C07325=1163.883,398.048,-85.044,-176.099,9.432,148.794
C07326=1163.887,397.800,-85.007,-176.099,9.430,148.793
C07327=1163.891,397.553,-84.971,-176.098,9.427,148.792
C07328=1163.895,397.306,-84.934,-176.097,9.426,148.792
C07329=1163.898,397.058,-84.899,-176.097,9.423,148.791
C07330=1163.903,396.811,-84.862,-176.097,9.420,148.790
C07331=1163.906,396.564,-84.826,-176.097,9.418,148.789
C07332=1163.910,396.316,-84.790,-176.096,9.416,148.789
C07333=1163.914,396.069,-84.754,-176.095,9.413,148.788
C07334=1163.918,395.822,-84.717,-176.095,9.410,148.787
C07335=1163.922,395.575,-84.680,-176.095,9.408,148.786
C07336=1163.926,395.327,-84.645,-176.094,9.406,148.785
C07337=1163.930,395.080,-84.608,-176.094,9.403,148.785
C07338=1163.934,394.832,-84.572,-176.094,9.401,148.784
C07339=1163.938,394.585,-84.535,-176.093,9.398,148.783
C07340=1163.941,394.338,-84.500,-176.093,9.395,148.782
C07341=1163.945,394.090,-84.463,-176.093,9.393,148.782
C07342=1163.949,393.843,-84.428,-176.092,9.390,148.781
C07343=1163.953,393.596,-84.391,-176.092,9.387,148.780
C07344=1163.957,393.349,-84.354,-176.091,9.385,148.779
C07345=1163.961,393.101,-84.318,-176.091,9.383,148.779
C07346=1163.964,392.854,-84.282,-176.091,9.379,148.778
C07347=1163.969,392.606,-84.246,-176.091,9.377,148.777
C07348=1163.972,392.359,-84.210,-176.091,9.374,148.776
C07349=1163.976,392.112,-84.173,-176.090,9.371,148.775
C07350=1163.980,391.827,-84.131,-176.090,9.368,148.775
C07351=1163.985,391.541,-84.090,-176.090,9.365,148.774
C07352=1163.990,391.256,-84.048,-176.089,9.362,148.773
C07353=1163.994,390.970,-84.006,-176.090,9.358,148.772
C07354=1163.998,390.723,-83.971,-176.089,9.355,148.771
C07355=1164.002,390.476,-83.934,-176.089,9.353,148.770
C07356=1164.006,390.228,-83.898,-176.089,9.349,148.770
C07357=1164.010,389.981,-83.861,-176.089,9.347,148.769
C07358=1164.013,389.733,-83.826,-176.089,9.344,148.768
C07359=1164.018,389.486,-83.789,-176.089,9.341,148.767
C07360=1164.021,389.239,-83.753,-176.089,9.338,148.766
C07361=1164.025,388.992,-83.717,-176.088,9.335,148.766
C07362=1164.029,388.744,-83.681,-176.089,9.332,148.765
C07363=1164.033,388.497,-83.644,-176.089,9.329,148.764
C07364=1164.037,388.249,-83.609,-176.089,9.326,148.763
C07365=1164.041,388.002,-83.572,-176.090,9.322,148.763
C07366=1164.044,387.755,-83.536,-176.089,9.320,148.762
C07367=1164.048,387.507,-83.501,-176.089,9.316,148.761
C07368=1164.052,387.260,-83.464,-176.090,9.313,148.760
C07369=1164.056,387.013,-83.428,-176.090,9.310,148.759
C07370=1164.060,386.765,-83.391,-176.090,9.307,148.759
C07371=1164.064,386.518,-83.356,-176.091,9.303,148.758
C07372=1164.068,386.270,-83.320,-176.091,9.300,148.757
C07373=1164.072,386.024,-83.284,-176.091,9.297,148.756
C07374=1164.076,385.776,-83.248,-176.091,9.294,148.756
C07375=1164.080,385.529,-83.211,-176.092,9.291,148.755
C07376=1164.083,385.282,-83.176,-176.092,9.287,148.754
C07377=1164.088,385.034,-83.140,-176.093,9.284,148.753
C07378=1164.091,384.787,-83.103,-176.093,9.281,148.753
C07379=1164.096,384.539,-83.067,-176.094,9.277,148.752
C07380=1164.099,384.292,-83.032,-176.094,9.274,148.751
C07381=1164.103,384.045,-82.996,-176.095,9.271,148.750
C07382=1164.107,383.797,-82.959,-176.096,9.266,148.750
C07383=1164.111,383.549,-82.924,-176.096,9.263,148.749
C07384=1164.114,383.303,-82.888,-176.097,9.260,148.748
C07385=1164.118,383.055,-82.851,-176.098,9.257,148.747
C07386=1164.123,382.808,-82.816,-176.099,9.252,148.747
C07387=1164.127,382.560,-82.780,-176.099,9.249,148.746
C07388=1164.130,382.313,-82.744,-176.100,9.246,148.745
C07389=1164.134,382.066,-82.708,-176.100,9.243,148.745
C07390=1164.139,381.818,-82.672,-176.101,9.238,148.744
C07391=1164.142,381.570,-82.637,-176.102,9.235,148.743
C07392=1164.146,381.324,-82.600,-176.103,9.231,148.742
C07393=1164.150,381.076,-82.564,-176.104,9.228,148.742
C07394=1164.154,380.828,-82.529,-176.105,9.224,148.741
C07395=1164.157,380.581,-82.493,-176.106,9.221,148.740
C07396=1164.162,380.334,-82.457,-176.107,9.217,148.740
C07397=1164.166,380.087,-82.421,-176.108,9.213,148.739
C07398=1164.169,379.839,-82.385,-176.109,9.209,148.738
C07399=1164.173,379.592,-82.350,-176.110,9.206,148.738
C07400=1164.177,379.344,-82.314,-176.111,9.202,148.737
C07401=1164.181,379.096,-82.278,-176.113,9.198,148.736
C07402=1164.185,378.849,-82.243,-176.113,9.195,148.736
C07403=1164.190,378.602,-82.207,-176.115,9.191,148.735
C07404=1164.193,378.355,-82.171,-176.116,9.187,148.734
C07405=1164.197,378.107,-82.135,-176.117,9.184,148.734
C07406=1164.200,377.860,-82.100,-176.118,9.180,148.733
C07407=1164.205,377.612,-82.063,-176.120,9.176,148.732
C07408=1164.208,377.365,-82.028,-176.121,9.172,148.732
C07409=1164.213,377.118,-81.993,-176.122,9.168,148.731
C07410=1164.216,376.870,-81.957,-176.123,9.165,148.731
C07411=1164.220,376.623,-81.922,-176.125,9.161,148.730
C07412=1164.224,376.375,-81.885,-176.126,9.157,148.729
C07413=1164.228,376.128,-81.850,-176.128,9.154,148.729
C07414=1164.232,375.881,-81.815,-176.129,9.150,148.728
C07415=1164.236,375.633,-81.779,-176.131,9.146,148.728
C07416=1164.240,375.386,-81.744,-176.132,9.142,148.727
C07417=1164.244,375.138,-81.707,-176.134,9.138,148.726
C07418=1164.248,374.890,-81.672,-176.136,9.135,148.726
C07419=1164.252,374.644,-81.637,-176.137,9.131,148.725
C07420=1164.256,374.396,-81.601,-176.138,9.127,148.725
C07421=1164.259,374.149,-81.566,-176.140,9.123,148.724
C07422=1164.263,373.901,-81.530,-176.142,9.119,148.724
C07423=1164.267,373.653,-81.495,-176.144,9.116,148.723
C07424=1164.272,373.406,-81.460,-176.145,9.112,148.723
C07425=1164.276,373.158,-81.424,-176.147,9.108,148.722
C07426=1164.279,372.911,-81.388,-176.148,9.104,148.722
C07427=1164.283,372.663,-81.353,-176.150,9.101,148.721
C07428=1164.287,372.417,-81.318,-176.152,9.097,148.721
C07429=1164.291,372.169,-81.282,-176.154,9.092,148.720
C07430=1164.295,371.921,-81.247,-176.156,9.089,148.720
C07431=1164.299,371.674,-81.212,-176.157,9.085,148.719
C07432=1164.303,371.427,-81.177,-176.159,9.081,148.719
C07433=1164.306,371.179,-81.141,-176.161,9.078,148.718
C07434=1164.310,370.931,-81.106,-176.163,9.073,148.717
C07435=1164.315,370.684,-81.071,-176.165,9.069,148.717
C07436=1164.318,370.437,-81.035,-176.167,9.066,148.717
C07437=1164.322,370.189,-81.000,-176.169,9.062,148.716
C07438=1164.327,369.942,-80.965,-176.171,9.059,148.716
C07439=1164.330,369.694,-80.930,-176.173,9.054,148.715
C07440=1164.334,369.447,-80.894,-176.175,9.051,148.715
C07441=1164.338,369.199,-80.860,-176.176,9.047,148.714
C07442=1164.342,368.952,-80.824,-176.179,9.042,148.714
C07443=1164.346,368.704,-80.789,-176.181,9.039,148.713
C07444=1164.350,368.456,-80.754,-176.182,9.035,148.713
C07445=1164.354,368.210,-80.719,-176.185,9.031,148.713
C07446=1164.358,367.961,-80.684,-176.187,9.027,148.712
C07447=1164.362,367.714,-80.648,-176.189,9.024,148.712
C07448=1164.366,367.467,-80.613,-176.191,9.019,148.711
C07449=1164.370,367.219,-80.578,-176.193,9.016,148.711
C07450=1164.374,366.972,-80.543,-176.195,9.012,148.710
C07451=1164.378,366.724,-80.508,-176.198,9.008,148.710
C07452=1164.382,366.477,-80.473,-176.200,9.004,148.710
C07453=1164.386,366.229,-80.438,-176.202,9.001,148.709
C07454=1164.391,365.947,-80.399,-176.204,8.996,148.709
C07455=1164.395,365.664,-80.359,-176.207,8.992,148.708
C07456=1164.399,365.382,-80.319,-176.209,8.988,148.708
C07457=1164.403,365.100,-80.279,-176.212,8.983,148.707
C07458=1164.407,364.852,-80.244,-176.214,8.979,148.707
C07459=1164.412,364.605,-80.209,-176.216,8.975,148.707
C07460=1164.416,364.357,-80.174,-176.219,8.971,148.706
C07461=1164.420,364.110,-80.139,-176.221,8.968,148.706
C07462=1164.423,363.862,-80.105,-176.223,8.964,148.706
C07463=1164.427,363.614,-80.070,-176.226,8.960,148.705
C07464=1164.431,363.367,-80.035,-176.228,8.956,148.705
C07465=1164.435,363.119,-80.000,-176.231,8.952,148.705
C07466=1164.440,362.872,-79.965,-176.232,8.949,148.704
C07467=1164.443,362.624,-79.931,-176.235,8.945,148.704
C07468=1164.447,362.377,-79.896,-176.237,8.941,148.704
C07469=1164.451,362.129,-79.861,-176.239,8.938,148.703
C07470=1164.455,361.881,-79.826,-176.242,8.933,148.703
C07471=1164.459,361.634,-79.792,-176.244,8.930,148.703
C07472=1164.463,361.386,-79.757,-176.247,8.926,148.702
C07473=1164.467,361.139,-79.723,-176.249,8.922,148.702
C07474=1164.471,360.891,-79.688,-176.251,8.918,148.701
C07475=1164.475,360.643,-79.654,-176.254,8.915,148.701
C07476=1164.479,360.396,-79.618,-176.256,8.910,148.701
C07477=1164.483,360.149,-79.584,-176.258,8.907,148.701
C07478=1164.487,359.901,-79.550,-176.261,8.904,148.700
C07479=1164.491,359.653,-79.515,-176.263,8.899,148.700
C07480=1164.494,359.406,-79.481,-176.265,8.896,148.700
C07481=1164.499,359.158,-79.446,-176.268,8.892,148.699
C07482=1164.503,358.910,-79.412,-176.270,8.888,148.699
C07483=1164.507,358.663,-79.378,-176.273,8.884,148.699
C07484=1164.511,358.415,-79.343,-176.275,8.881,148.698
C07485=1164.515,358.168,-79.309,-176.277,8.877,148.698
C07486=1164.519,357.921,-79.274,-176.280,8.873,148.698
C07487=1164.523,357.673,-79.239,-176.282,8.870,148.698
C07488=1164.527,357.426,-79.205,-176.285,8.866,148.697
C07489=1164.531,357.178,-79.170,-176.287,8.862,148.697
C07490=1164.535,356.930,-79.137,-176.289,8.859,148.697
C07491=1164.539,356.682,-79.102,-176.292,8.855,148.696
C07492=1164.543,356.435,-79.068,-176.294,8.851,148.696
C07493=1164.547,356.187,-79.034,-176.297,8.847,148.696
C07494=1164.550,355.939,-79.000,-176.299,8.844,148.695
C07495=1164.555,355.692,-78.965,-176.302,8.840,148.695
C07496=1164.558,355.444,-78.931,-176.304,8.836,148.695
C07497=1164.563,355.197,-78.897,-176.306,8.833,148.695
C07498=1164.567,354.950,-78.863,-176.309,8.829,148.694
C07499=1164.571,354.701,-78.828,-176.311,8.825,148.694
C07500=1164.575,354.454,-78.795,-176.313,8.822,148.694
C07501=1164.579,354.206,-78.760,-176.316,8.817,148.693
C07502=1164.583,353.958,-78.726,-176.318,8.814,148.693
C07503=1164.587,353.711,-78.692,-176.321,8.811,148.693
C07504=1164.590,353.463,-78.657,-176.323,8.806,148.693
C07505=1164.595,353.215,-78.624,-176.325,8.803,148.692
C07506=1164.599,352.968,-78.590,-176.328,8.800,148.692
C07507=1164.602,352.720,-78.555,-176.331,8.796,148.692
C07508=1164.607,352.473,-78.521,-176.333,8.792,148.692
C07509=1164.611,352.225,-78.488,-176.335,8.789,148.691
C07510=1164.615,351.977,-78.453,-176.338,8.785,148.691
C07511=1164.619,351.730,-78.419,-176.340,8.781,148.691
C07512=1164.623,351.482,-78.386,-176.342,8.778,148.690
C07513=1164.627,351.235,-78.351,-176.345,8.774,148.690
C07514=1164.631,350.987,-78.317,-176.347,8.771,148.690
C07515=1164.635,350.739,-78.284,-176.350,8.766,148.690
C07516=1164.639,350.492,-78.250,-176.352,8.763,148.689
C07517=1164.643,350.243,-78.216,-176.354,8.760,148.689
C07518=1164.647,349.996,-78.182,-176.357,8.756,148.689
C07519=1164.652,349.748,-78.148,-176.360,8.752,148.689
C07520=1164.656,349.501,-78.115,-176.362,8.749,148.688
C07521=1164.659,349.253,-78.080,-176.365,8.745,148.688
C07522=1164.664,349.005,-78.047,-176.367,8.742,148.688
C07523=1164.667,348.758,-78.013,-176.369,8.738,148.688
C07524=1164.672,348.510,-77.980,-176.372,8.734,148.687
C07525=1164.676,348.262,-77.945,-176.374,8.731,148.687
C07526=1164.680,348.015,-77.912,-176.376,8.727,148.687
C07527=1164.684,347.767,-77.878,-176.379,8.724,148.687
C07528=1164.688,347.520,-77.845,-176.382,8.720,148.686
C07529=1164.691,347.271,-77.811,-176.384,8.717,148.686
C07530=1164.696,347.024,-77.777,-176.386,8.713,148.686
C07531=1164.700,346.776,-77.743,-176.389,8.709,148.686
C07532=1164.704,346.528,-77.710,-176.391,8.706,148.685
C07533=1164.708,346.281,-77.676,-176.394,8.703,148.685
C07534=1164.712,346.033,-77.642,-176.396,8.699,148.685
C07535=1164.716,345.785,-77.608,-176.399,8.695,148.685
C07536=1164.720,345.538,-77.575,-176.401,8.692,148.685
C07537=1164.724,345.290,-77.542,-176.403,8.688,148.684
C07538=1164.728,345.042,-77.509,-176.406,8.684,148.684
C07539=1164.732,344.795,-77.475,-176.408,8.681,148.684
C07540=1164.736,344.547,-77.442,-176.410,8.678,148.684
C07541=1164.741,344.299,-77.408,-176.413,8.674,148.683
C07542=1164.745,344.051,-77.375,-176.416,8.670,148.683
C07543=1164.749,343.804,-77.341,-176.418,8.667,148.683
C07544=1164.753,343.556,-77.308,-176.421,8.663,148.683
C07545=1164.757,343.308,-77.274,-176.423,8.660,148.682
C07546=1164.761,343.061,-77.241,-176.425,8.656,148.682
C07547=1164.765,342.813,-77.208,-176.428,8.652,148.682
C07548=1164.768,342.565,-77.174,-176.430,8.649,148.682
C07549=1164.773,342.317,-77.141,-176.433,8.646,148.681
C07550=1164.777,342.070,-77.108,-176.435,8.642,148.681
C07551=1164.781,341.822,-77.074,-176.438,8.638,148.681
C07552=1164.786,341.574,-77.041,-176.441,8.635,148.681
C07553=1164.790,341.326,-77.008,-176.443,8.632,148.681
C07554=1164.794,341.078,-76.974,-176.445,8.629,148.681
C07555=1164.798,340.831,-76.941,-176.448,8.624,148.680
C07556=1164.802,340.583,-76.908,-176.450,8.621,148.680
C07557=1164.806,340.335,-76.875,-176.453,8.618,148.680
C07558=1164.811,340.056,-76.837,-176.456,8.614,148.680
C07559=1164.815,339.776,-76.800,-176.458,8.610,148.679
C07560=1164.819,339.497,-76.763,-176.461,8.606,148.679
C07561=1164.824,339.217,-76.725,-176.464,8.602,148.679
C07562=1164.828,338.970,-76.692,-176.466,8.598,148.679
C07563=1164.832,338.722,-76.659,-176.469,8.595,148.678
C07564=1164.836,338.474,-76.626,-176.471,8.592,148.678
C07565=1164.841,338.226,-76.593,-176.474,8.587,148.678
C07566=1164.845,337.979,-76.560,-176.476,8.584,148.678
C07567=1164.849,337.730,-76.527,-176.479,8.581,148.678
C07568=1164.853,337.483,-76.494,-176.481,8.578,148.678
C07569=1164.857,337.235,-76.461,-176.484,8.574,148.677
C07570=1164.861,336.987,-76.428,-176.486,8.570,148.677
C07571=1164.865,336.740,-76.395,-176.489,8.567,148.677
C07572=1164.869,336.492,-76.362,-176.491,8.564,148.677
C07573=1164.874,336.244,-76.330,-176.493,8.561,148.677
C07574=1164.878,335.996,-76.296,-176.496,8.556,148.676
C07575=1164.882,335.748,-76.263,-176.499,8.553,148.676
C07576=1164.885,335.501,-76.231,-176.501,8.550,148.676
C07577=1164.890,335.252,-76.198,-176.503,8.547,148.676
C07578=1164.894,335.005,-76.165,-176.506,8.543,148.676
C07579=1164.898,334.757,-76.132,-176.509,8.540,148.675
C07580=1164.901,334.509,-76.099,-176.511,8.536,148.675
C07581=1164.906,334.261,-76.067,-176.513,8.533,148.675
C07582=1164.910,334.013,-76.034,-176.517,8.529,148.675
C07583=1164.914,333.766,-76.001,-176.519,8.526,148.675
C07584=1164.918,333.518,-75.969,-176.521,8.523,148.675
C07585=1164.922,333.270,-75.936,-176.523,8.519,148.674
C07586=1164.926,333.022,-75.902,-176.526,8.516,148.674
C07587=1164.931,332.774,-75.870,-176.529,8.512,148.674
C07588=1164.935,332.527,-75.838,-176.531,8.509,148.674
C07589=1164.939,332.279,-75.805,-176.534,8.506,148.674
C07590=1164.943,332.031,-75.772,-176.536,8.502,148.674
C07591=1164.947,331.783,-75.740,-176.539,8.498,148.673
C07592=1164.951,331.535,-75.707,-176.541,8.495,148.673
C07593=1164.955,331.287,-75.675,-176.544,8.492,148.673
C07594=1164.959,331.039,-75.642,-176.546,8.489,148.673
C07595=1164.963,330.791,-75.610,-176.548,8.485,148.673
C07596=1164.967,330.543,-75.577,-176.551,8.481,148.672
C07597=1164.972,330.296,-75.545,-176.554,8.478,148.672
C07598=1164.976,330.048,-75.512,-176.556,8.475,148.672
C07599=1164.980,329.800,-75.480,-176.559,8.472,148.672
C07600=1164.984,329.553,-75.447,-176.561,8.468,148.672
C07601=1164.988,329.304,-75.415,-176.564,8.464,148.672
C07602=1164.991,329.057,-75.382,-176.566,8.461,148.672
C07603=1164.997,328.809,-75.350,-176.569,8.458,148.671
C07604=1165.001,328.561,-75.317,-176.571,8.455,148.671
C07605=1165.004,328.313,-75.285,-176.573,8.451,148.671
C07606=1165.009,328.065,-75.252,-176.577,8.448,148.671
C07607=1165.013,327.817,-75.221,-176.579,8.444,148.671
C07608=1165.017,327.570,-75.188,-176.581,8.441,148.671
C07609=1165.021,327.322,-75.156,-176.584,8.438,148.670
C07610=1165.025,327.074,-75.124,-176.586,8.435,148.670
C07611=1165.029,326.826,-75.091,-176.589,8.431,148.670
C07612=1165.033,326.578,-75.059,-176.591,8.427,148.670
C07613=1165.038,326.330,-75.027,-176.594,8.424,148.670
C07614=1165.042,326.082,-74.995,-176.597,8.421,148.670
C07615=1165.046,325.834,-74.963,-176.599,8.418,148.670
C07616=1165.050,325.586,-74.930,-176.601,8.414,148.669
C07617=1165.054,325.339,-74.898,-176.604,8.412,148.669
C07618=1165.059,325.091,-74.866,-176.607,8.407,148.669
C07619=1165.062,324.843,-74.834,-176.609,8.404,148.669
C07620=1165.066,324.595,-74.802,-176.612,8.401,148.669
C07621=1165.071,324.347,-74.770,-176.614,8.398,148.669
C07622=1165.074,324.100,-74.737,-176.616,8.395,148.668
C07623=1165.079,323.851,-74.705,-176.619,8.392,148.668
C07624=1165.083,323.603,-74.673,-176.622,8.387,148.668
C07625=1165.087,323.356,-74.642,-176.624,8.384,148.668
C07626=1165.091,323.107,-74.609,-176.627,8.381,148.668
C07627=1165.095,322.859,-74.577,-176.629,8.378,148.668
C07628=1165.099,322.612,-74.546,-176.632,8.375,148.668
C07629=1165.104,322.364,-74.513,-176.634,8.372,148.668
C07630=1165.108,322.116,-74.482,-176.637,8.368,148.667
C07631=1165.111,321.868,-74.450,-176.639,8.364,148.667
C07632=1165.116,321.620,-74.418,-176.642,8.361,148.667
C07633=1165.120,321.372,-74.386,-176.644,8.358,148.667
C07634=1165.124,321.124,-74.354,-176.647,8.355,148.667
C07635=1165.129,320.876,-74.322,-176.650,8.352,148.667
C07636=1165.132,320.628,-74.290,-176.652,8.348,148.667
C07637=1165.136,320.380,-74.258,-176.655,8.344,148.666
C07638=1165.140,320.133,-74.227,-176.657,8.341,148.666
C07639=1165.145,319.885,-74.194,-176.660,8.338,148.666
C07640=1165.149,319.636,-74.162,-176.662,8.335,148.666
C07641=1165.153,319.389,-74.132,-176.665,8.332,148.666
C07642=1165.157,319.140,-74.100,-176.667,8.328,148.666
C07643=1165.162,318.893,-74.068,-176.670,8.326,148.666
C07644=1165.166,318.645,-74.036,-176.673,8.321,148.666
C07645=1165.169,318.397,-74.004,-176.675,8.318,148.665
C07646=1165.174,318.149,-73.973,-176.678,8.315,148.665
C07647=1165.178,317.901,-73.941,-176.680,8.312,148.665
C07648=1165.183,317.653,-73.909,-176.683,8.309,148.665
C07649=1165.186,317.405,-73.878,-176.685,8.306,148.665
C07650=1165.190,317.157,-73.846,-176.687,8.302,148.665
C07651=1165.195,316.909,-73.815,-176.690,8.299,148.665
C07652=1165.198,316.661,-73.783,-176.693,8.295,148.665
C07653=1165.203,316.414,-73.752,-176.696,8.292,148.665
C07654=1165.208,316.165,-73.720,-176.698,8.289,148.665
C07655=1165.212,315.917,-73.688,-176.700,8.286,148.664
C07656=1165.216,315.669,-73.657,-176.703,8.283,148.664
C07657=1165.220,315.421,-73.625,-176.705,8.279,148.664
C07658=1165.224,315.173,-73.594,-176.708,8.276,148.664
C07659=1165.228,314.925,-73.562,-176.710,8.273,148.664
C07660=1165.232,314.677,-73.531,-176.714,8.269,148.664
C07661=1165.236,314.429,-73.499,-176.716,8.266,148.664
C07662=1165.241,314.152,-73.464,-176.719,8.263,148.664
C07663=1165.246,313.875,-73.430,-176.722,8.259,148.664
C07664=1165.250,313.598,-73.394,-176.724,8.256,148.664
C07665=1165.255,313.321,-73.359,-176.727,8.252,148.663
C07666=1165.259,313.073,-73.329,-176.729,8.249,148.663
C07667=1165.263,312.825,-73.297,-176.732,8.246,148.663
C07668=1165.267,312.577,-73.266,-176.734,8.242,148.663
C07669=1165.271,312.329,-73.234,-176.737,8.239,148.663
C07670=1165.276,312.081,-73.203,-176.740,8.235,148.663
C07671=1165.280,311.833,-73.172,-176.743,8.232,148.663
C07672=1165.284,311.585,-73.141,-176.745,8.229,148.663
C07673=1165.288,311.337,-73.109,-176.748,8.226,148.663
C07674=1165.292,311.089,-73.078,-176.750,8.223,148.662
C07675=1165.296,310.840,-73.047,-176.753,8.220,148.662
C07676=1165.301,310.593,-73.016,-176.755,8.216,148.662
C07677=1165.305,310.345,-72.985,-176.758,8.213,148.662
C07678=1165.309,310.096,-72.954,-176.760,8.210,148.662
C07679=1165.314,309.849,-72.922,-176.763,8.207,148.662
C07680=1165.318,309.600,-72.891,-176.765,8.204,148.662
C07681=1165.322,309.352,-72.860,-176.769,8.200,148.662
C07682=1165.326,309.104,-72.829,-176.771,8.197,148.662
C07683=1165.331,308.857,-72.798,-176.774,8.194,148.662
C07684=1165.335,308.609,-72.767,-176.776,8.191,148.662
C07685=1165.339,308.360,-72.736,-176.779,8.188,148.662
C07686=1165.343,308.113,-72.705,-176.781,8.184,148.661
C07687=1165.347,307.865,-72.674,-176.784,8.181,148.661
C07688=1165.351,307.616,-72.643,-176.786,8.178,148.661
C07689=1165.356,307.368,-72.612,-176.789,8.175,148.661
C07690=1165.360,307.120,-72.581,-176.791,8.172,148.661
C07691=1165.364,306.873,-72.550,-176.794,8.169,148.661
C07692=1165.368,306.625,-72.520,-176.796,8.165,148.661
C07693=1165.372,306.376,-72.488,-176.799,8.163,148.661
C07694=1165.377,306.128,-72.458,-176.801,8.159,148.661
C07695=1165.382,305.880,-72.427,-176.804,8.155,148.661
C07696=1165.385,305.632,-72.396,-176.807,8.152,148.661
C07697=1165.389,305.384,-72.366,-176.809,8.149,148.660
C07698=1165.394,305.136,-72.335,-176.812,8.146,148.661
C07699=1165.398,304.888,-72.303,-176.814,8.143,148.660
C07700=1165.402,304.640,-72.273,-176.817,8.140,148.660
C07701=1165.406,304.392,-72.242,-176.820,8.137,148.660
C07702=1165.410,304.143,-72.211,-176.822,8.134,148.660
C07703=1165.415,303.896,-72.180,-176.825,8.130,148.660
C07704=1165.419,303.648,-72.150,-176.827,8.127,148.660
C07705=1165.423,303.400,-72.119,-176.830,8.124,148.660
C07706=1165.427,303.151,-72.088,-176.832,8.121,148.660
C07707=1165.431,302.904,-72.058,-176.835,8.118,148.660
C07708=1165.436,302.655,-72.028,-176.837,8.115,148.660
C07709=1165.441,302.407,-71.997,-176.840,8.112,148.660
C07710=1165.444,302.159,-71.967,-176.842,8.109,148.660
C07711=1165.449,301.911,-71.936,-176.845,8.106,148.660
C07712=1165.453,301.663,-71.905,-176.848,8.103,148.660
C07713=1165.457,301.415,-71.875,-176.850,8.099,148.659
C07714=1165.461,301.167,-71.844,-176.853,8.096,148.659
C07715=1165.466,300.919,-71.813,-176.856,8.092,148.659
C07716=1165.470,300.670,-71.784,-176.859,8.089,148.659
C07717=1165.475,300.422,-71.753,-176.861,8.086,148.659
C07718=1165.478,300.174,-71.722,-176.864,8.083,148.659
C07719=1165.482,299.926,-71.691,-176.866,8.080,148.659
C07720=1165.486,299.678,-71.661,-176.869,8.077,148.659
C07721=1165.491,299.430,-71.631,-176.871,8.074,148.659
C07722=1165.496,299.182,-71.600,-176.874,8.071,148.659
C07723=1165.499,298.933,-71.570,-176.876,8.068,148.659
C07724=1165.504,298.686,-71.539,-176.879,8.065,148.659
C07725=1165.508,298.437,-71.510,-176.882,8.062,148.659
C07726=1165.513,298.189,-71.479,-176.884,8.058,148.659
C07727=1165.516,297.942,-71.449,-176.887,8.055,148.659
C07728=1165.521,297.692,-71.418,-176.889,8.052,148.659
C07729=1165.525,297.445,-71.388,-176.892,8.049,148.659
C07730=1165.529,297.197,-71.357,-176.895,8.046,148.659
C07731=1165.533,296.949,-71.328,-176.897,8.043,148.658
C07732=1165.538,296.701,-71.297,-176.900,8.040,148.658
C07733=1165.542,296.453,-71.267,-176.903,8.037,148.658
C07734=1165.545,296.204,-71.237,-176.905,8.034,148.658
C07735=1165.550,295.956,-71.206,-176.908,8.031,148.658
C07736=1165.554,295.708,-71.177,-176.910,8.028,148.658
C07737=1165.559,295.460,-71.146,-176.913,8.024,148.658
C07738=1165.563,295.211,-71.117,-176.915,8.021,148.658
C07739=1165.567,294.964,-71.087,-176.918,8.019,148.658
C07740=1165.572,294.715,-71.057,-176.920,8.015,148.658
C07741=1165.576,294.468,-71.026,-176.923,8.012,148.658
C07742=1165.581,294.219,-70.996,-176.926,8.009,148.658
C07743=1165.584,293.971,-70.966,-176.928,8.006,148.658
C07744=1165.588,293.722,-70.936,-176.931,8.003,148.658
C07745=1165.593,293.474,-70.906,-176.934,8.000,148.658
C07746=1165.597,293.226,-70.876,-176.936,7.997,148.658
C07747=1165.601,292.979,-70.846,-176.939,7.994,148.658
C07748=1165.606,292.730,-70.816,-176.941,7.991,148.658
C07749=1165.610,292.482,-70.787,-176.944,7.988,148.658
C07750=1165.614,292.234,-70.756,-176.947,7.985,148.658
C07751=1165.618,291.986,-70.727,-176.949,7.982,148.658
C07752=1165.623,291.738,-70.696,-176.952,7.978,148.658
C07753=1165.627,291.490,-70.667,-176.954,7.975,148.658
C07754=1165.631,291.241,-70.637,-176.957,7.972,148.658
C07755=1165.635,290.993,-70.608,-176.960,7.969,148.658
C07756=1165.640,290.745,-70.577,-176.962,7.966,148.658
C07757=1165.644,290.497,-70.548,-176.965,7.963,148.658
C07758=1165.648,290.249,-70.518,-176.968,7.960,148.658
C07759=1165.652,290.001,-70.488,-176.970,7.957,148.657
C07760=1165.657,289.752,-70.458,-176.973,7.954,148.657
C07761=1165.661,289.504,-70.428,-176.975,7.951,148.658
C07762=1165.665,289.256,-70.399,-176.978,7.948,148.658
C07763=1165.669,289.008,-70.370,-176.980,7.945,148.657
C07764=1165.673,288.760,-70.339,-176.983,7.942,148.657
C07765=1165.678,288.511,-70.309,-176.986,7.939,148.657
C07766=1165.682,288.236,-70.277,-176.989,7.936,148.657
C07767=1165.687,287.961,-70.244,-176.991,7.933,148.657
C07768=1165.692,287.686,-70.211,-176.994,7.929,148.657
C07769=1165.697,287.411,-70.178,-176.997,7.926,148.657
C07770=1165.701,287.163,-70.149,-177.000,7.923,148.657
C07771=1165.705,286.915,-70.119,-177.003,7.920,148.657
C07772=1165.709,286.667,-70.090,-177.005,7.917,148.657
C07773=1165.713,286.418,-70.060,-177.008,7.914,148.657
C07774=1165.718,286.170,-70.030,-177.010,7.911,148.657
C07775=1165.722,285.921,-70.001,-177.013,7.908,148.657
C07776=1165.727,285.674,-69.972,-177.015,7.904,148.657
C07777=1165.731,285.426,-69.942,-177.018,7.901,148.657
C07778=1165.736,285.177,-69.913,-177.021,7.898,148.657
C07779=1165.740,284.929,-69.883,-177.024,7.895,148.657
C07780=1165.744,284.681,-69.854,-177.026,7.892,148.657
C07781=1165.748,284.432,-69.824,-177.029,7.889,148.657
C07782=1165.752,284.184,-69.795,-177.031,7.886,148.657
C07783=1165.756,283.936,-69.765,-177.034,7.883,148.657
C07784=1165.761,283.688,-69.736,-177.037,7.880,148.657
C07785=1165.765,283.440,-69.707,-177.039,7.877,148.657
C07786=1165.770,283.192,-69.677,-177.041,7.875,148.657
C07787=1165.774,282.944,-69.648,-177.044,7.872,148.657
C07788=1165.778,282.695,-69.619,-177.047,7.869,148.657
C07789=1165.782,282.446,-69.590,-177.050,7.866,148.657
C07790=1165.787,282.198,-69.560,-177.052,7.863,148.657
C07791=1165.791,281.950,-69.531,-177.055,7.860,148.657
C07792=1165.796,281.702,-69.502,-177.057,7.857,148.657
C07793=1165.800,281.454,-69.472,-177.060,7.854,148.657
C07794=1165.804,281.205,-69.444,-177.063,7.851,148.657
C07795=1165.808,280.957,-69.414,-177.065,7.848,148.657
C07796=1165.813,280.709,-69.385,-177.068,7.845,148.657
C07797=1165.817,280.461,-69.356,-177.071,7.842,148.657
C07798=1165.821,280.213,-69.328,-177.073,7.839,148.657
C07799=1165.825,279.964,-69.298,-177.076,7.836,148.657
C07800=1165.830,279.716,-69.269,-177.078,7.834,148.657
C07801=1165.834,279.467,-69.240,-177.081,7.830,148.657
C07802=1165.839,279.220,-69.211,-177.083,7.827,148.657
C07803=1165.843,278.971,-69.181,-177.086,7.824,148.657
C07804=1165.847,278.723,-69.153,-177.089,7.821,148.657
C07805=1165.851,278.474,-69.124,-177.092,7.818,148.657
C07806=1165.855,278.226,-69.094,-177.094,7.815,148.657
C07807=1165.860,277.978,-69.066,-177.097,7.812,148.657
C07808=1165.864,277.730,-69.036,-177.099,7.809,148.657
C07809=1165.868,277.481,-69.008,-177.102,7.806,148.657
C07810=1165.872,277.233,-68.979,-177.105,7.803,148.657
C07811=1165.877,276.985,-68.950,-177.108,7.800,148.657
C07812=1165.882,276.736,-68.921,-177.110,7.798,148.658
C07813=1165.885,276.488,-68.892,-177.113,7.795,148.658
C07814=1165.890,276.240,-68.863,-177.115,7.792,148.658
C07815=1165.894,275.992,-68.834,-177.118,7.789,148.657
C07816=1165.899,275.743,-68.806,-177.120,7.786,148.657
C07817=1165.902,275.495,-68.777,-177.123,7.783,148.658
C07818=1165.907,275.247,-68.748,-177.126,7.780,148.658
C07819=1165.911,274.999,-68.719,-177.129,7.777,148.658
C07820=1165.916,274.750,-68.690,-177.131,7.774,148.658
C07821=1165.920,274.502,-68.662,-177.134,7.772,148.658
C07822=1165.925,274.254,-68.633,-177.136,7.769,148.658
C07823=1165.929,274.005,-68.604,-177.139,7.766,148.658
C07824=1165.933,273.758,-68.576,-177.141,7.763,148.658
C07825=1165.938,273.509,-68.547,-177.144,7.760,148.658
C07826=1165.942,273.260,-68.518,-177.147,7.757,148.658
C07827=1165.946,273.012,-68.490,-177.150,7.754,148.658
C07828=1165.951,272.764,-68.461,-177.152,7.751,148.658
C07829=1165.954,272.515,-68.433,-177.155,7.748,148.658
C07830=1165.959,272.267,-68.404,-177.157,7.746,148.658
C07831=1165.964,272.019,-68.375,-177.160,7.743,148.658
C07832=1165.967,271.770,-68.347,-177.163,7.740,148.658
C07833=1165.972,271.522,-68.318,-177.166,7.737,148.658
C07834=1165.976,271.274,-68.290,-177.168,7.734,148.658
C07835=1165.981,271.026,-68.261,-177.171,7.731,148.658
C07836=1165.985,270.777,-68.233,-177.173,7.728,148.658
C07837=1165.989,270.528,-68.204,-177.176,7.725,148.658
C07838=1165.994,270.281,-68.175,-177.178,7.723,148.658
C07839=1165.998,270.032,-68.147,-177.181,7.720,148.658
C07840=1166.003,269.784,-68.119,-177.184,7.717,148.658
C07841=1166.007,269.535,-68.091,-177.187,7.714,148.658
C07842=1166.011,269.286,-68.062,-177.189,7.711,148.658
C07843=1166.015,269.039,-68.034,-177.192,7.708,148.658
C07844=1166.020,268.790,-68.005,-177.195,7.705,148.659
C07845=1166.024,268.542,-67.977,-177.197,7.703,148.659
C07846=1166.028,268.293,-67.948,-177.200,7.700,148.659
C07847=1166.033,268.046,-67.920,-177.203,7.697,148.659
C07848=1166.037,267.797,-67.892,-177.205,7.694,148.659
C07849=1166.042,267.549,-67.864,-177.208,7.691,148.659
C07850=1166.046,267.300,-67.835,-177.211,7.688,148.659
C07851=1166.050,267.052,-67.807,-177.214,7.685,148.659
C07852=1166.054,266.804,-67.779,-177.216,7.683,148.659
C07853=1166.059,266.555,-67.751,-177.219,7.680,148.659
C07854=1166.063,266.307,-67.723,-177.221,7.677,148.659
C07855=1166.068,266.058,-67.694,-177.224,7.674,148.659
C07856=1166.072,265.810,-67.666,-177.227,7.671,148.659
C07857=1166.076,265.562,-67.638,-177.230,7.668,148.659
C07858=1166.081,265.313,-67.610,-177.232,7.666,148.659
C07859=1166.085,265.065,-67.582,-177.234,7.663,148.659
C07860=1166.090,264.816,-67.553,-177.237,7.660,148.659
C07861=1166.094,264.569,-67.525,-177.240,7.657,148.659
C07862=1166.098,264.319,-67.498,-177.242,7.654,148.659
C07863=1166.103,264.071,-67.470,-177.245,7.651,148.659
C07864=1166.107,263.823,-67.441,-177.247,7.649,148.660
C07865=1166.111,263.575,-67.414,-177.250,7.646,148.660
C07866=1166.116,263.326,-67.385,-177.253,7.643,148.660
C07867=1166.120,263.078,-67.357,-177.256,7.640,148.660
C07868=1166.124,262.829,-67.330,-177.259,7.637,148.660
C07869=1166.128,262.581,-67.302,-177.261,7.635,148.660
C07870=1166.134,262.307,-67.271,-177.264,7.631,148.660
C07871=1166.138,262.034,-67.240,-177.267,7.628,148.660
C07872=1166.143,261.762,-67.209,-177.270,7.625,148.660
C07873=1166.148,261.489,-67.178,-177.273,7.622,148.660
C07874=1166.152,261.239,-67.151,-177.275,7.619,148.660
C07875=1166.156,260.992,-67.123,-177.278,7.616,148.660
C07876=1166.161,260.744,-67.095,-177.281,7.613,148.660
C07877=1166.166,260.494,-67.067,-177.283,7.611,148.660
C07878=1166.170,260.246,-67.040,-177.286,7.608,148.661
C07879=1166.174,259.998,-67.011,-177.288,7.605,148.661
C07880=1166.178,259.749,-66.984,-177.291,7.602,148.661
C07881=1166.183,259.501,-66.957,-177.294,7.599,148.661
C07882=1166.186,259.253,-66.928,-177.296,7.597,148.661
C07883=1166.192,259.004,-66.901,-177.299,7.595,148.661
C07884=1166.196,258.756,-66.873,-177.302,7.592,148.661
C07885=1166.200,258.507,-66.846,-177.305,7.589,148.661
C07886=1166.205,258.259,-66.818,-177.308,7.586,148.661
C07887=1166.209,258.011,-66.790,-177.310,7.584,148.661
C07888=1166.213,257.762,-66.763,-177.313,7.581,148.661
C07889=1166.217,257.514,-66.735,-177.315,7.578,148.661
C07890=1166.222,257.266,-66.708,-177.318,7.575,148.662
C07891=1166.227,257.017,-66.679,-177.321,7.572,148.662
C07892=1166.231,256.768,-66.652,-177.323,7.570,148.662
C07893=1166.236,256.520,-66.624,-177.326,7.567,148.662
C07894=1166.240,256.271,-66.597,-177.329,7.564,148.662
C07895=1166.244,256.023,-66.569,-177.331,7.561,148.662
C07896=1166.249,255.775,-66.542,-177.334,7.559,148.662
C07897=1166.253,255.526,-66.515,-177.337,7.556,148.662
C07898=1166.257,255.278,-66.487,-177.339,7.553,148.662
C07899=1166.262,255.029,-66.460,-177.342,7.550,148.662
C07900=1166.266,254.781,-66.432,-177.345,7.547,148.662
C07901=1166.270,254.532,-66.404,-177.347,7.545,148.663
C07902=1166.275,254.284,-66.377,-177.350,7.542,148.663
C07903=1166.279,254.036,-66.350,-177.353,7.539,148.663
C07904=1166.284,253.787,-66.323,-177.355,7.536,148.663
C07905=1166.288,253.538,-66.295,-177.358,7.534,148.663
C07906=1166.292,253.290,-66.267,-177.361,7.531,148.663
C07907=1166.297,253.042,-66.240,-177.364,7.529,148.663
C07908=1166.301,252.793,-66.213,-177.366,7.526,148.663
C07909=1166.306,252.544,-66.186,-177.369,7.523,148.663
C07910=1166.310,252.296,-66.158,-177.371,7.520,148.663
C07911=1166.315,252.048,-66.131,-177.374,7.518,148.663
C07912=1166.319,251.799,-66.104,-177.377,7.515,148.663
C07913=1166.323,251.551,-66.077,-177.380,7.513,148.664
C07914=1166.327,251.302,-66.049,-177.382,7.510,148.664
C07915=1166.332,251.054,-66.022,-177.385,7.507,148.664
C07916=1166.336,250.805,-65.995,-177.388,7.504,148.664
C07917=1166.341,250.557,-65.968,-177.390,7.502,148.664
C07918=1166.345,250.308,-65.941,-177.393,7.499,148.664
C07919=1166.350,250.060,-65.914,-177.396,7.496,148.664
C07920=1166.354,249.811,-65.886,-177.399,7.493,148.664
C07921=1166.358,249.563,-65.859,-177.401,7.491,148.665
C07922=1166.362,249.315,-65.832,-177.404,7.488,148.665
C07923=1166.367,249.066,-65.805,-177.406,7.485,148.665
C07924=1166.372,248.818,-65.778,-177.409,7.483,148.665
C07925=1166.376,248.569,-65.751,-177.412,7.480,148.665
C07926=1166.380,248.320,-65.724,-177.415,7.477,148.665
C07927=1166.384,248.072,-65.697,-177.417,7.475,148.665
C07928=1166.389,247.823,-65.670,-177.420,7.472,148.665
C07929=1166.394,247.575,-65.643,-177.422,7.469,148.665
C07930=1166.398,247.326,-65.616,-177.425,7.466,148.665
C07931=1166.402,247.078,-65.590,-177.428,7.464,148.666
C07932=1166.407,246.830,-65.562,-177.430,7.462,148.666
C07933=1166.412,246.581,-65.535,-177.433,7.459,148.666
C07934=1166.416,246.333,-65.508,-177.436,7.456,148.666
C07935=1166.420,246.084,-65.482,-177.438,7.454,148.666
C07936=1166.424,245.835,-65.454,-177.441,7.451,148.666
C07937=1166.429,245.587,-65.427,-177.444,7.448,148.666
C07938=1166.433,245.338,-65.401,-177.446,7.446,148.667
C07939=1166.437,245.090,-65.374,-177.449,7.443,148.667
C07940=1166.442,244.841,-65.348,-177.452,7.440,148.667
C07941=1166.446,244.593,-65.321,-177.455,7.437,148.667
C07942=1166.451,244.344,-65.294,-177.457,7.435,148.667
C07943=1166.456,244.096,-65.267,-177.460,7.432,148.667
C07944=1166.460,243.848,-65.240,-177.463,7.429,148.667
C07945=1166.464,243.599,-65.213,-177.465,7.428,148.668
C07946=1166.469,243.350,-65.187,-177.468,7.425,148.668
C07947=1166.473,243.102,-65.161,-177.471,7.422,148.668
C07948=1166.478,242.853,-65.134,-177.473,7.420,148.668
C07949=1166.482,242.605,-65.106,-177.476,7.417,148.668
C07950=1166.487,242.356,-65.081,-177.479,7.414,148.668
C07951=1166.491,242.107,-65.054,-177.481,7.412,148.668
C07952=1166.495,241.859,-65.027,-177.484,7.409,148.668
C07953=1166.500,241.611,-65.000,-177.487,7.406,148.669
C07954=1166.504,241.362,-64.974,-177.490,7.404,148.669
C07955=1166.509,241.113,-64.947,-177.492,7.401,148.669
C07956=1166.513,240.865,-64.920,-177.495,7.398,148.669
C07957=1166.518,240.616,-64.895,-177.498,7.396,148.669
C07958=1166.522,240.368,-64.867,-177.500,7.394,148.669
C07959=1166.526,240.119,-64.841,-177.503,7.391,148.669
C07960=1166.531,239.870,-64.815,-177.505,7.388,148.669
C07961=1166.535,239.622,-64.788,-177.509,7.386,148.670
C07962=1166.540,239.373,-64.762,-177.511,7.383,148.670
C07963=1166.544,239.125,-64.735,-177.514,7.381,148.670
C07964=1166.549,238.876,-64.709,-177.516,7.378,148.670
C07965=1166.553,238.628,-64.683,-177.520,7.375,148.670
C07966=1166.558,238.379,-64.655,-177.522,7.373,148.670
C07967=1166.562,238.130,-64.630,-177.525,7.370,148.670
C07968=1166.566,237.882,-64.603,-177.528,7.367,148.671
C07969=1166.571,237.634,-64.577,-177.530,7.365,148.671
C07970=1166.575,237.386,-64.551,-177.533,7.362,148.671
C07971=1166.580,237.136,-64.524,-177.536,7.360,148.671
C07972=1166.584,236.888,-64.498,-177.538,7.358,148.671
C07973=1166.589,236.639,-64.472,-177.541,7.355,148.671
C07974=1166.593,236.368,-64.443,-177.544,7.352,148.672
C07975=1166.598,236.096,-64.415,-177.547,7.349,148.672
C07976=1166.603,235.824,-64.386,-177.550,7.346,148.672
C07977=1166.608,235.552,-64.357,-177.553,7.344,148.672
C07978=1166.613,235.304,-64.330,-177.555,7.341,148.672
C07979=1166.617,235.055,-64.305,-177.558,7.339,148.672
C07980=1166.621,234.806,-64.279,-177.561,7.336,148.673
C07981=1166.626,234.558,-64.252,-177.563,7.334,148.673
C07982=1166.630,234.310,-64.226,-177.566,7.331,148.673
C07983=1166.635,234.061,-64.201,-177.569,7.328,148.673
C07984=1166.639,233.812,-64.174,-177.571,7.326,148.673
C07985=1166.644,233.564,-64.148,-177.574,7.323,148.673
C07986=1166.648,233.315,-64.122,-177.577,7.321,148.674
C07987=1166.653,233.067,-64.097,-177.580,7.318,148.674
C07988=1166.657,232.818,-64.070,-177.582,7.315,148.674
C07989=1166.662,232.569,-64.044,-177.585,7.314,148.674
C07990=1166.666,232.321,-64.018,-177.588,7.311,148.674
C07991=1166.671,232.071,-63.992,-177.591,7.308,148.674
C07992=1166.675,231.824,-63.966,-177.593,7.306,148.675
C07993=1166.679,231.575,-63.940,-177.596,7.303,148.675
C07994=1166.684,231.326,-63.914,-177.599,7.301,148.675
C07995=1166.688,231.078,-63.889,-177.601,7.298,148.675
C07996=1166.693,230.828,-63.862,-177.604,7.295,148.675
C07997=1166.698,230.580,-63.837,-177.607,7.294,148.675
C07998=1166.702,230.332,-63.810,-177.610,7.291,148.675
C07999=1166.706,230.083,-63.785,-177.612,7.288,148.676
C08000=1166.710,229.835,-63.759,-177.615,7.286,148.676
C08001=1166.716,229.586,-63.733,-177.617,7.284,148.676
C08002=1166.720,229.337,-63.707,-177.620,7.281,148.676
C08003=1166.724,229.089,-63.681,-177.623,7.278,148.676
C08004=1166.728,228.840,-63.656,-177.625,7.276,148.677
C08005=1166.733,228.592,-63.630,-177.629,7.273,148.677
C08006=1166.737,228.343,-63.604,-177.631,7.271,148.677
C08007=1166.742,228.094,-63.579,-177.634,7.269,148.677
C08008=1166.747,227.846,-63.553,-177.637,7.266,148.677
C08009=1166.751,227.597,-63.527,-177.639,7.264,148.677
C08010=1166.756,227.348,-63.501,-177.642,7.261,148.678
C08011=1166.760,227.099,-63.475,-177.644,7.259,148.678
C08012=1166.765,226.851,-63.450,-177.647,7.256,148.678
C08013=1166.769,226.602,-63.424,-177.650,7.254,148.678
C08014=1166.773,226.353,-63.399,-177.653,7.251,148.678
C08015=1166.778,226.105,-63.373,-177.656,7.249,148.679
C08016=1166.782,225.857,-63.347,-177.658,7.246,148.679
C08017=1166.786,225.608,-63.322,-177.661,7.244,148.679
C08018=1166.791,225.360,-63.296,-177.664,7.242,148.679
C08019=1166.796,225.110,-63.271,-177.666,7.239,148.679
C08020=1166.800,224.861,-63.246,-177.669,7.237,148.680
C08021=1166.805,224.613,-63.220,-177.672,7.234,148.680
C08022=1166.809,224.365,-63.194,-177.674,7.232,148.680
C08023=1166.814,224.116,-63.169,-177.677,7.229,148.680
C08024=1166.818,223.868,-63.143,-177.680,7.227,148.680
C08025=1166.823,223.618,-63.118,-177.683,7.225,148.680
C08026=1166.827,223.370,-63.093,-177.685,7.222,148.681
C08027=1166.832,223.121,-63.067,-177.688,7.220,148.681
C08028=1166.836,222.872,-63.041,-177.691,7.217,148.681
C08029=1166.841,222.624,-63.017,-177.693,7.215,148.681
C08030=1166.845,222.375,-62.991,-177.696,7.212,148.681
C08031=1166.850,222.127,-62.966,-177.699,7.210,148.682
C08032=1166.854,221.878,-62.940,-177.702,7.207,148.682
C08033=1166.859,221.629,-62.915,-177.704,7.206,148.682
C08034=1166.864,221.380,-62.889,-177.707,7.203,148.682
C08035=1166.868,221.132,-62.864,-177.709,7.201,148.682
C08036=1166.872,220.883,-62.840,-177.713,7.198,148.683
C08037=1166.876,220.634,-62.814,-177.715,7.196,148.683
C08038=1166.881,220.386,-62.788,-177.718,7.193,148.683
C08039=1166.886,220.137,-62.763,-177.720,7.191,148.683
C08040=1166.890,219.888,-62.738,-177.723,7.189,148.684
C08041=1166.895,219.639,-62.713,-177.726,7.186,148.684
C08042=1166.899,219.391,-62.688,-177.729,7.184,148.684
C08043=1166.903,219.143,-62.662,-177.731,7.182,148.684
C08044=1166.908,218.893,-62.637,-177.734,7.179,148.684
C08045=1166.913,218.645,-62.612,-177.736,7.177,148.684
C08046=1166.917,218.396,-62.587,-177.740,7.174,148.685
C08047=1166.922,218.148,-62.562,-177.742,7.172,148.685
C08048=1166.926,217.899,-62.537,-177.745,7.170,148.685
C08049=1166.931,217.651,-62.512,-177.747,7.167,148.685
C08050=1166.935,217.401,-62.487,-177.751,7.165,148.686
C08051=1166.940,217.153,-62.461,-177.753,7.163,148.686
C08052=1166.944,216.904,-62.437,-177.756,7.160,148.686
C08053=1166.949,216.656,-62.411,-177.758,7.158,148.686
C08054=1166.953,216.406,-62.386,-177.761,7.155,148.686
C08055=1166.958,216.158,-62.362,-177.764,7.153,148.687
C08056=1166.962,215.909,-62.337,-177.767,7.151,148.687
C08057=1166.967,215.660,-62.312,-177.769,7.149,148.687
C08058=1166.971,215.412,-62.286,-177.772,7.146,148.687
C08059=1166.976,215.163,-62.262,-177.774,7.144,148.687
C08060=1166.980,214.914,-62.237,-177.778,7.141,148.688
C08061=1166.985,214.666,-62.212,-177.780,7.139,148.688
C08062=1166.989,214.417,-62.188,-177.783,7.137,148.688
C08063=1166.994,214.168,-62.163,-177.785,7.134,148.688
C08064=1166.999,213.920,-62.137,-177.789,7.132,148.689
C08065=1167.003,213.671,-62.113,-177.791,7.130,148.689
C08066=1167.008,213.422,-62.088,-177.794,7.127,148.689
C08067=1167.012,213.173,-62.062,-177.796,7.125,148.689
C08068=1167.016,212.925,-62.038,-177.799,7.122,148.689
C08069=1167.021,212.676,-62.014,-177.802,7.120,148.690
C08070=1167.025,212.427,-61.989,-177.804,7.118,148.690
C08071=1167.030,212.179,-61.964,-177.807,7.115,148.690
C08072=1167.035,211.929,-61.939,-177.810,7.114,148.690
C08073=1167.039,211.681,-61.915,-177.813,7.111,148.690
C08074=1167.044,211.432,-61.890,-177.815,7.109,148.691
C08075=1167.048,211.183,-61.866,-177.818,7.106,148.691
C08076=1167.053,210.935,-61.840,-177.821,7.104,148.691
C08077=1167.057,210.687,-61.816,-177.824,7.102,148.692
C08078=1167.062,210.416,-61.789,-177.826,7.100,148.692
C08079=1167.067,210.145,-61.763,-177.829,7.097,148.692
C08080=1167.072,209.875,-61.736,-177.833,7.094,148.692
C08081=1167.077,209.604,-61.709,-177.835,7.091,148.692
C08082=1167.082,209.355,-61.685,-177.838,7.090,148.693
C08083=1167.086,209.106,-61.660,-177.841,7.088,148.693
C08084=1167.091,208.857,-61.635,-177.843,7.085,148.693
C08085=1167.095,208.610,-61.611,-177.846,7.083,148.694
C08086=1167.100,208.361,-61.586,-177.849,7.080,148.694
C08087=1167.104,208.112,-61.562,-177.852,7.078,148.694
C08088=1167.109,207.863,-61.537,-177.854,7.075,148.694
C08089=1167.113,207.615,-61.513,-177.857,7.074,148.694
C08090=1167.118,207.365,-61.488,-177.860,7.072,148.695
C08091=1167.122,207.117,-61.464,-177.862,7.069,148.695
C08092=1167.128,206.868,-61.439,-177.865,7.067,148.695
C08093=1167.132,206.618,-61.415,-177.868,7.064,148.695
C08094=1167.136,206.370,-61.391,-177.871,7.062,148.696
C08095=1167.141,206.121,-61.367,-177.873,7.060,148.696
C08096=1167.146,205.873,-61.342,-177.876,7.058,148.696
C08097=1167.150,205.623,-61.317,-177.879,7.056,148.696
C08098=1167.154,205.375,-61.293,-177.881,7.053,148.697
C08099=1167.159,205.126,-61.269,-177.884,7.051,148.697
C08100=1167.164,204.878,-61.245,-177.886,7.049,148.697
C08101=1167.168,204.629,-61.220,-177.890,7.047,148.697
C08102=1167.172,204.380,-61.196,-177.892,7.045,148.698
C08103=1167.178,204.131,-61.172,-177.895,7.042,148.698
C08104=1167.182,203.882,-61.148,-177.898,7.040,148.698
C08105=1167.186,203.634,-61.124,-177.900,7.038,148.698
C08106=1167.191,203.385,-61.099,-177.903,7.035,148.699
C08107=1167.195,203.136,-61.075,-177.906,7.034,148.699
C08108=1167.200,202.887,-61.052,-177.909,7.031,148.699
C08109=1167.205,202.638,-61.027,-177.911,7.029,148.699
C08110=1167.209,202.389,-61.002,-177.914,7.027,148.700
C08111=1167.213,202.141,-60.978,-177.917,7.024,148.700
C08112=1167.218,201.892,-60.955,-177.919,7.022,148.700
C08113=1167.223,201.643,-60.930,-177.922,7.019,148.700
C08114=1167.228,201.395,-60.906,-177.925,7.018,148.701
C08115=1167.232,201.146,-60.883,-177.928,7.016,148.701
C08116=1167.236,200.897,-60.858,-177.930,7.013,148.701
C08117=1167.240,200.648,-60.834,-177.933,7.011,148.701
C08118=1167.246,200.399,-60.810,-177.936,7.009,148.702
C08119=1167.250,200.150,-60.786,-177.938,7.006,148.702
C08120=1167.255,199.902,-60.762,-177.941,7.005,148.702
C08121=1167.259,199.653,-60.739,-177.943,7.003,148.702
C08122=1167.263,199.404,-60.714,-177.947,7.000,148.703
C08123=1167.268,199.155,-60.690,-177.949,6.998,148.703
C08124=1167.273,198.906,-60.666,-177.952,6.995,148.703
C08125=1167.277,198.658,-60.642,-177.955,6.993,148.703
C08126=1167.282,198.409,-60.619,-177.957,6.992,148.704
C08127=1167.287,198.160,-60.595,-177.960,6.989,148.704
C08128=1167.291,197.911,-60.572,-177.963,6.987,148.704
C08129=1167.296,197.662,-60.547,-177.965,6.985,148.705
C08130=1167.301,197.413,-60.524,-177.968,6.982,148.705
C08131=1167.305,197.164,-60.499,-177.971,6.981,148.705
C08132=1167.310,196.915,-60.476,-177.974,6.979,148.705
C08133=1167.314,196.667,-60.452,-177.976,6.976,148.705
C08134=1167.319,196.418,-60.428,-177.979,6.974,148.706
C08135=1167.323,196.169,-60.404,-177.982,6.972,148.706
C08136=1167.328,195.920,-60.381,-177.984,6.969,148.706
C08137=1167.332,195.672,-60.357,-177.987,6.968,148.707
C08138=1167.337,195.423,-60.333,-177.990,6.966,148.707
C08139=1167.342,195.174,-60.310,-177.993,6.963,148.707
C08140=1167.346,194.926,-60.286,-177.995,6.961,148.707
C08141=1167.351,194.677,-60.263,-177.998,6.959,148.708
C08142=1167.356,194.428,-60.238,-178.001,6.956,148.708
C08143=1167.360,194.179,-60.215,-178.003,6.955,148.708
C08144=1167.365,193.930,-60.191,-178.006,6.953,148.709
C08145=1167.370,193.681,-60.167,-178.009,6.950,148.709
C08146=1167.374,193.432,-60.144,-178.012,6.948,148.709
C08147=1167.379,193.183,-60.121,-178.014,6.946,148.709
C08148=1167.383,192.935,-60.096,-178.017,6.944,148.710
C08149=1167.387,192.686,-60.074,-178.020,6.942,148.710
C08150=1167.392,192.437,-60.050,-178.022,6.940,148.710
C08151=1167.397,192.188,-60.027,-178.026,6.937,148.711
C08152=1167.401,191.940,-60.003,-178.028,6.935,148.711
C08153=1167.406,191.691,-59.980,-178.031,6.933,148.711
C08154=1167.410,191.442,-59.956,-178.033,6.932,148.711
C08155=1167.415,191.193,-59.933,-178.036,6.929,148.712
C08156=1167.420,190.943,-59.909,-178.039,6.927,148.712
C08157=1167.424,190.695,-59.885,-178.041,6.925,148.712
C08158=1167.429,190.446,-59.862,-178.045,6.923,148.713
C08159=1167.434,190.197,-59.839,-178.047,6.920,148.713
C08160=1167.438,189.948,-59.815,-178.049,6.919,148.713
C08161=1167.443,189.699,-59.792,-178.053,6.916,148.713
C08162=1167.447,189.450,-59.769,-178.055,6.914,148.714
C08163=1167.451,189.202,-59.745,-178.058,6.912,148.714
C08164=1167.456,188.953,-59.722,-178.060,6.910,148.714
C08165=1167.461,188.704,-59.698,-178.064,6.908,148.715
C08166=1167.466,188.455,-59.675,-178.066,6.906,148.715
C08167=1167.471,188.206,-59.652,-178.068,6.904,148.715
C08168=1167.476,187.957,-59.629,-178.072,6.901,148.715
C08169=1167.479,187.709,-59.606,-178.074,6.900,148.716
C08170=1167.484,187.460,-59.583,-178.077,6.898,148.716
C08171=1167.489,187.211,-59.559,-178.079,6.896,148.716
C08172=1167.494,186.962,-59.536,-178.082,6.893,148.717
C08173=1167.498,186.713,-59.512,-178.085,6.891,148.717
C08174=1167.502,186.464,-59.490,-178.087,6.889,148.717
C08175=1167.508,186.215,-59.467,-178.090,6.888,148.717
C08176=1167.512,185.966,-59.443,-178.093,6.885,148.718
C08177=1167.517,185.717,-59.420,-178.096,6.883,148.718
C08178=1167.521,185.469,-59.397,-178.098,6.881,148.718
C08179=1167.526,185.220,-59.374,-178.101,6.878,148.719
C08180=1167.530,184.971,-59.351,-178.104,6.877,148.719
C08181=1167.534,184.722,-59.328,-178.107,6.875,148.719
C08182=1167.540,184.452,-59.303,-178.110,6.872,148.720
C08183=1167.545,184.182,-59.278,-178.113,6.871,148.720
C08184=1167.549,183.913,-59.253,-178.116,6.868,148.720
C08185=1167.555,183.643,-59.228,-178.118,6.866,148.720
C08186=1167.560,183.394,-59.205,-178.121,6.864,148.721
C08187=1167.564,183.146,-59.182,-178.124,6.862,148.721
C08188=1167.569,182.897,-59.159,-178.127,6.860,148.722
C08189=1167.574,182.647,-59.136,-178.129,6.858,148.722
C08190=1167.578,182.399,-59.114,-178.132,6.856,148.722
C08191=1167.582,182.150,-59.090,-178.135,6.853,148.722
C08192=1167.588,181.901,-59.067,-178.138,6.852,148.723
C08193=1167.592,181.653,-59.045,-178.140,6.850,148.723
C08194=1167.597,181.403,-59.022,-178.143,6.848,148.723
C08195=1167.601,181.154,-58.999,-178.145,6.846,148.724
C08196=1167.606,180.906,-58.976,-178.148,6.843,148.724
C08197=1167.611,180.657,-58.953,-178.151,6.842,148.724
C08198=1167.615,180.408,-58.931,-178.154,6.840,148.725
C08199=1167.620,180.158,-58.907,-178.156,6.838,148.725
C08200=1167.624,179.910,-58.885,-178.159,6.835,148.725
C08201=1167.629,179.661,-58.862,-178.162,6.833,148.725
C08202=1167.633,179.412,-58.840,-178.165,6.832,148.726
C08203=1167.638,179.163,-58.816,-178.167,6.830,148.726
C08204=1167.643,178.914,-58.794,-178.170,6.828,148.726
C08205=1167.647,178.665,-58.771,-178.173,6.825,148.727
C08206=1167.652,178.416,-58.748,-178.176,6.823,148.727
C08207=1167.656,178.167,-58.726,-178.178,6.822,148.727
C08208=1167.662,177.919,-58.703,-178.181,6.820,148.728
C08209=1167.666,177.669,-58.681,-178.184,6.817,148.728
C08210=1167.671,177.420,-58.657,-178.186,6.815,148.728
C08211=1167.676,177.172,-58.636,-178.189,6.813,148.729
C08212=1167.680,176.923,-58.612,-178.192,6.812,148.729
C08213=1167.685,176.673,-58.590,-178.194,6.810,148.729
C08214=1167.689,176.425,-58.568,-178.198,6.807,148.730
C08215=1167.694,176.176,-58.545,-178.200,6.805,148.730
C08216=1167.698,175.927,-58.522,-178.203,6.803,148.730
C08217=1167.704,175.678,-58.500,-178.205,6.802,148.731
C08218=1167.708,175.429,-58.477,-178.208,6.800,148.731
C08219=1167.713,175.180,-58.455,-178.211,6.798,148.731
C08220=1167.717,174.932,-58.432,-178.214,6.796,148.732
C08221=1167.721,174.682,-58.410,-178.216,6.794,148.732
C08222=1167.726,174.433,-58.387,-178.219,6.792,148.732
C08223=1167.731,174.185,-58.365,-178.221,6.790,148.732
C08224=1167.736,173.936,-58.342,-178.224,6.788,148.733
C08225=1167.740,173.686,-58.320,-178.227,6.786,148.733
C08226=1167.745,173.438,-58.298,-178.230,6.784,148.734
C08227=1167.750,173.188,-58.275,-178.233,6.782,148.734
C08228=1167.754,172.940,-58.253,-178.235,6.780,148.734
C08229=1167.759,172.691,-58.231,-178.238,6.778,148.734
C08230=1167.763,172.441,-58.208,-178.240,6.777,148.735
C08231=1167.768,172.193,-58.186,-178.244,6.774,148.735
C08232=1167.773,171.943,-58.164,-178.246,6.772,148.736
C08233=1167.778,171.695,-58.141,-178.249,6.770,148.736
C08234=1167.782,171.446,-58.119,-178.252,6.769,148.736
C08235=1167.786,171.196,-58.097,-178.254,6.767,148.736
C08236=1167.792,170.948,-58.075,-178.257,6.765,148.737
C08237=1167.796,170.699,-58.052,-178.260,6.762,148.737
C08238=1167.801,170.450,-58.030,-178.263,6.760,148.737
C08239=1167.805,170.201,-58.008,-178.265,6.759,148.738
C08240=1167.811,169.952,-57.986,-178.268,6.757,148.738
C08241=1167.815,169.703,-57.963,-178.271,6.755,148.739
C08242=1167.820,169.455,-57.941,-178.273,6.753,148.739
C08243=1167.824,169.205,-57.919,-178.275,6.751,148.739
C08244=1167.829,168.956,-57.897,-178.279,6.749,148.739
C08245=1167.834,168.707,-57.875,-178.281,6.747,148.740
C08246=1167.838,168.458,-57.852,-178.284,6.745,148.740
C08247=1167.842,168.210,-57.831,-178.287,6.743,148.741
C08248=1167.847,167.960,-57.808,-178.289,6.742,148.741
C08249=1167.852,167.711,-57.786,-178.292,6.740,148.741
C08250=1167.857,167.462,-57.764,-178.295,6.738,148.742
C08251=1167.861,167.213,-57.743,-178.298,6.736,148.742
C08252=1167.866,166.964,-57.721,-178.300,6.734,148.742
C08253=1167.871,166.715,-57.699,-178.303,6.732,148.743
C08254=1167.876,166.466,-57.677,-178.306,6.730,148.743
C08255=1167.881,166.217,-57.655,-178.308,6.728,148.743
C08256=1167.885,165.968,-57.633,-178.311,6.727,148.744
C08257=1167.890,165.719,-57.611,-178.314,6.725,148.744
C08258=1167.895,165.470,-57.589,-178.316,6.723,148.744
C08259=1167.899,165.221,-57.567,-178.319,6.721,148.745
C08260=1167.904,164.972,-57.545,-178.322,6.719,148.745
C08261=1167.908,164.723,-57.523,-178.325,6.717,148.745
C08262=1167.913,164.474,-57.502,-178.328,6.715,148.746
C08263=1167.918,164.225,-57.479,-178.330,6.713,148.746
C08264=1167.923,163.976,-57.457,-178.333,6.711,148.746
C08265=1167.927,163.727,-57.435,-178.335,6.710,148.747
C08266=1167.932,163.478,-57.414,-178.338,6.708,148.747
C08267=1167.937,163.229,-57.392,-178.341,6.706,148.747
C08268=1167.941,162.980,-57.370,-178.343,6.704,148.748
C08269=1167.946,162.732,-57.348,-178.346,6.703,148.748
C08270=1167.950,162.482,-57.326,-178.349,6.700,148.749
C08271=1167.955,162.234,-57.304,-178.352,6.698,148.749
C08272=1167.960,161.984,-57.283,-178.355,6.696,148.749
C08273=1167.964,161.735,-57.261,-178.358,6.695,148.750
C08274=1167.969,161.486,-57.240,-178.360,6.693,148.750
C08275=1167.974,161.237,-57.218,-178.363,6.691,148.750
C08276=1167.978,160.988,-57.196,-178.366,6.689,148.751
C08277=1167.983,160.740,-57.174,-178.368,6.688,148.751
C08278=1167.988,160.490,-57.153,-178.370,6.686,148.751
C08279=1167.993,160.241,-57.131,-178.373,6.684,148.752
C08280=1167.998,159.992,-57.110,-178.376,6.682,148.752
C08281=1168.002,159.743,-57.088,-178.379,6.680,148.752
C08282=1168.007,159.494,-57.067,-178.382,6.678,148.753
C08283=1168.011,159.245,-57.046,-178.385,6.676,148.753
C08284=1168.015,158.996,-57.023,-178.387,6.674,148.754
C08285=1168.020,158.748,-57.002,-178.390,6.673,148.754
C08286=1168.026,158.478,-56.978,-178.393,6.671,148.754
C08287=1168.031,158.209,-56.956,-178.395,6.669,148.755
C08288=1168.036,157.940,-56.932,-178.399,6.667,148.755
C08289=1168.040,157.671,-56.909,-178.402,6.665,148.756
C08290=1168.046,157.422,-56.888,-178.404,6.663,148.756
C08291=1168.050,157.173,-56.866,-178.407,6.662,148.756
C08292=1168.055,156.924,-56.844,-178.410,6.660,148.757
C08293=1168.060,156.675,-56.823,-178.413,6.658,148.757
C08294=1168.065,156.426,-56.802,-178.415,6.656,148.757
C08295=1168.069,156.177,-56.781,-178.417,6.654,148.758
C08296=1168.074,155.928,-56.759,-178.420,6.652,148.758
C08297=1168.078,155.679,-56.737,-178.423,6.651,148.758
C08298=1168.084,155.430,-56.716,-178.426,6.649,148.759
C08299=1168.088,155.181,-56.694,-178.429,6.646,148.759
C08300=1168.092,154.932,-56.674,-178.431,6.645,148.760
C08301=1168.097,154.683,-56.652,-178.434,6.643,148.760
C08302=1168.102,154.434,-56.631,-178.437,6.641,148.760
C08303=1168.107,154.184,-56.609,-178.440,6.639,148.761
C08304=1168.112,153.935,-56.588,-178.442,6.638,148.761
C08305=1168.116,153.687,-56.567,-178.445,6.636,148.761
C08306=1168.121,153.438,-56.546,-178.448,6.634,148.762
C08307=1168.125,153.188,-56.524,-178.450,6.632,148.762
C08308=1168.130,152.939,-56.503,-178.453,6.631,148.763
C08309=1168.135,152.691,-56.482,-178.456,6.629,148.763
C08310=1168.140,152.441,-56.461,-178.458,6.627,148.763
C08311=1168.145,152.192,-56.440,-178.461,6.625,148.764
C08312=1168.149,151.943,-56.418,-178.464,6.624,148.764
C08313=1168.154,151.694,-56.398,-178.467,6.622,148.764
C08314=1168.159,151.445,-56.376,-178.469,6.620,148.765
C08315=1168.164,151.196,-56.355,-178.472,6.618,148.765
C08316=1168.168,150.947,-56.335,-178.475,6.617,148.766
C08317=1168.172,150.698,-56.313,-178.477,6.615,148.766
C08318=1168.178,150.448,-56.292,-178.480,6.613,148.766
C08319=1168.182,150.199,-56.271,-178.483,6.612,148.767
C08320=1168.187,149.951,-56.250,-178.485,6.610,148.767
C08321=1168.192,149.702,-56.229,-178.488,6.608,148.767
C08322=1168.197,149.453,-56.208,-178.491,6.607,148.768
C08323=1168.201,149.204,-56.187,-178.494,6.605,148.768
C08324=1168.205,148.954,-56.166,-178.497,6.603,148.769
C08325=1168.210,148.705,-56.145,-178.499,6.601,148.769
C08326=1168.216,148.456,-56.124,-178.502,6.600,148.770
C08327=1168.220,148.207,-56.103,-178.505,6.598,148.770
C08328=1168.225,147.958,-56.082,-178.507,6.596,148.770
C08329=1168.229,147.709,-56.062,-178.510,6.594,148.771
C08330=1168.234,147.460,-56.041,-178.513,6.593,148.771
C08331=1168.239,147.210,-56.019,-178.516,6.591,148.772
C08332=1168.243,146.962,-55.998,-178.518,6.589,148.772
C08333=1168.248,146.712,-55.977,-178.521,6.587,148.772
C08334=1168.253,146.464,-55.957,-178.524,6.586,148.773
C08335=1168.258,146.214,-55.936,-178.526,6.584,148.773
C08336=1168.262,145.965,-55.916,-178.529,6.582,148.773
C08337=1168.268,145.716,-55.895,-178.532,6.580,148.774
C08338=1168.272,145.467,-55.874,-178.534,6.579,148.774
C08339=1168.277,145.218,-55.853,-178.537,6.577,148.775
C08340=1168.281,144.970,-55.832,-178.540,6.575,148.775
C08341=1168.287,144.720,-55.811,-178.543,6.574,148.775
C08342=1168.291,144.471,-55.791,-178.545,6.572,148.776
C08343=1168.296,144.222,-55.770,-178.548,6.570,148.776
C08344=1168.300,143.972,-55.749,-178.551,6.569,148.777
C08345=1168.305,143.723,-55.728,-178.554,6.567,148.777
C08346=1168.310,143.474,-55.708,-178.556,6.565,148.778
C08347=1168.315,143.225,-55.687,-178.559,6.564,148.778
C08348=1168.319,142.976,-55.666,-178.561,6.562,148.778
C08349=1168.324,142.727,-55.646,-178.564,6.561,148.779
C08350=1168.329,142.478,-55.625,-178.567,6.559,148.779
C08351=1168.333,142.229,-55.605,-178.569,6.557,148.779
C08352=1168.338,141.980,-55.584,-178.572,6.556,148.780
C08353=1168.343,141.731,-55.563,-178.575,6.554,148.780
C08354=1168.347,141.482,-55.543,-178.578,6.552,148.781
C08355=1168.352,141.232,-55.522,-178.580,6.550,148.781
C08356=1168.357,140.983,-55.502,-178.583,6.549,148.781
C08357=1168.362,140.734,-55.481,-178.586,6.547,148.782
C08358=1168.367,140.485,-55.460,-178.589,6.545,148.782
C08359=1168.371,140.236,-55.441,-178.591,6.544,148.783
C08360=1168.376,139.986,-55.420,-178.594,6.542,148.783
C08361=1168.381,139.737,-55.399,-178.597,6.540,148.784
C08362=1168.385,139.489,-55.379,-178.600,6.539,148.784
C08363=1168.390,139.239,-55.358,-178.602,6.537,148.784
C08364=1168.395,138.990,-55.338,-178.604,6.536,148.785
C08365=1168.399,138.741,-55.317,-178.607,6.534,148.785
C08366=1168.405,138.492,-55.297,-178.610,6.532,148.785
C08367=1168.410,138.243,-55.277,-178.613,6.531,148.786
C08368=1168.414,137.994,-55.257,-178.615,6.529,148.786
C08369=1168.419,137.745,-55.236,-178.618,6.528,148.787
C08370=1168.424,137.495,-55.216,-178.621,6.526,148.787
C08371=1168.429,137.246,-55.196,-178.624,6.524,148.788
C08372=1168.433,136.998,-55.175,-178.627,6.522,148.788
C08373=1168.438,136.748,-55.154,-178.629,6.521,148.788
C08374=1168.443,136.499,-55.135,-178.632,6.519,148.789
C08375=1168.447,136.250,-55.114,-178.635,6.517,148.789
C08376=1168.452,136.001,-55.094,-178.637,6.516,148.790
C08377=1168.456,135.752,-55.074,-178.639,6.514,148.790
C08378=1168.462,135.503,-55.054,-178.643,6.513,148.791
C08379=1168.467,135.254,-55.033,-178.645,6.511,148.791
C08380=1168.471,135.005,-55.013,-178.648,6.510,148.791
C08381=1168.476,134.755,-54.993,-178.651,6.508,148.792
C08382=1168.480,134.506,-54.973,-178.653,6.506,148.792
C08383=1168.486,134.256,-54.953,-178.656,6.504,148.793
C08384=1168.490,134.007,-54.932,-178.659,6.503,148.793
C08385=1168.495,133.759,-54.912,-178.662,6.501,148.793
C08386=1168.500,133.510,-54.893,-178.664,6.500,148.794
C08387=1168.505,133.261,-54.872,-178.667,6.499,148.794
C08388=1168.509,133.011,-54.853,-178.670,6.497,148.795
C08389=1168.515,132.762,-54.832,-178.672,6.495,148.795
C08390=1168.519,132.493,-54.811,-178.675,6.493,148.796
C08391=1168.525,132.225,-54.788,-178.678,6.492,148.796
C08392=1168.530,131.956,-54.767,-178.681,6.490,148.797
C08393=1168.535,131.688,-54.746,-178.684,6.489,148.797
C08394=1168.540,131.438,-54.725,-178.686,6.487,148.797
C08395=1168.545,131.189,-54.706,-178.689,6.485,148.798
C08396=1168.550,130.940,-54.685,-178.692,6.484,148.798
C08397=1168.554,130.691,-54.666,-178.695,6.482,148.799
C08398=1168.559,130.442,-54.645,-178.698,6.480,148.799
C08399=1168.563,130.192,-54.626,-178.700,6.479,148.800
C08400=1168.569,129.944,-54.606,-178.703,6.477,148.800
C08401=1168.573,129.695,-54.586,-178.705,6.476,148.800
C08402=1168.578,129.446,-54.566,-178.708,6.475,148.801
C08403=1168.582,129.196,-54.546,-178.711,6.473,148.801
C08404=1168.587,128.946,-54.526,-178.714,6.471,148.802
C08405=1168.592,128.698,-54.506,-178.716,6.469,148.802
C08406=1168.597,128.449,-54.487,-178.719,6.468,148.803
C08407=1168.602,128.199,-54.467,-178.722,6.466,148.803
C08408=1168.606,127.950,-54.447,-178.724,6.465,148.804
C08409=1168.611,127.701,-54.427,-178.727,6.464,148.804
C08410=1168.616,127.452,-54.407,-178.730,6.462,148.804
C08411=1168.621,127.203,-54.387,-178.733,6.460,148.805
C08412=1168.626,126.954,-54.368,-178.735,6.458,148.805
C08413=1168.631,126.704,-54.348,-178.738,6.457,148.806
C08414=1168.635,126.455,-54.328,-178.741,6.456,148.806
C08415=1168.640,126.206,-54.308,-178.743,6.454,148.807
C08416=1168.645,125.957,-54.289,-178.746,6.453,148.807
C08417=1168.650,125.708,-54.269,-178.749,6.451,148.807
C08418=1168.654,125.458,-54.249,-178.751,6.449,148.808
C08419=1168.660,125.210,-54.230,-178.754,6.447,148.808
C08420=1168.664,124.960,-54.211,-178.757,6.447,148.809
C08421=1168.668,124.711,-54.190,-178.759,6.445,148.809
C08422=1168.673,124.462,-54.171,-178.762,6.443,148.810
C08423=1168.678,124.213,-54.151,-178.765,6.442,148.810
C08424=1168.683,123.963,-54.132,-178.768,6.440,148.810
C08425=1168.688,123.714,-54.112,-178.771,6.439,148.811
C08426=1168.693,123.465,-54.093,-178.773,6.438,148.811
C08427=1168.698,123.216,-54.072,-178.776,6.436,148.812
C08428=1168.702,122.967,-54.053,-178.778,6.434,148.812
C08429=1168.707,122.718,-54.034,-178.781,6.432,148.813
C08430=1168.712,122.468,-54.014,-178.784,6.431,148.813
C08431=1168.717,122.219,-53.995,-178.786,6.430,148.814
C08432=1168.722,121.970,-53.975,-178.789,6.428,148.814
C08433=1168.727,121.720,-53.956,-178.792,6.427,148.814
C08434=1168.731,121.472,-53.937,-178.794,6.425,148.815
C08435=1168.736,121.222,-53.917,-178.798,6.424,148.815
C08436=1168.740,120.973,-53.897,-178.800,6.423,148.816
C08437=1168.746,120.724,-53.878,-178.802,6.421,148.816
C08438=1168.750,120.475,-53.858,-178.805,6.419,148.817
C08439=1168.755,120.226,-53.839,-178.808,6.418,148.817
C08440=1168.760,119.977,-53.820,-178.811,6.416,148.818
C08441=1168.764,119.727,-53.800,-178.813,6.415,148.818
C08442=1168.770,119.478,-53.781,-178.816,6.414,148.818
C08443=1168.774,119.229,-53.762,-178.819,6.412,148.819
C08444=1168.779,118.980,-53.742,-178.821,6.410,148.819
C08445=1168.784,118.731,-53.723,-178.825,6.409,148.820
C08446=1168.789,118.481,-53.703,-178.827,6.408,148.820
C08447=1168.793,118.232,-53.684,-178.829,6.406,148.821
C08448=1168.798,117.982,-53.665,-178.832,6.404,148.821
C08449=1168.804,117.733,-53.646,-178.835,6.403,148.822
C08450=1168.808,117.484,-53.627,-178.837,6.402,148.822
C08451=1168.813,117.235,-53.608,-178.840,6.400,148.823
C08452=1168.818,116.986,-53.588,-178.843,6.399,148.823
C08453=1168.822,116.737,-53.569,-178.846,6.397,148.824
C08454=1168.827,116.488,-53.550,-178.849,6.396,148.824
C08455=1168.832,116.239,-53.531,-178.851,6.395,148.824
C08456=1168.836,115.989,-53.511,-178.854,6.393,148.825
C08457=1168.842,115.740,-53.493,-178.856,6.391,148.825
C08458=1168.847,115.490,-53.473,-178.860,6.390,148.826
C08459=1168.851,115.242,-53.455,-178.862,6.389,148.826
C08460=1168.856,114.992,-53.435,-178.864,6.387,148.827
C08461=1168.862,114.743,-53.416,-178.867,6.386,148.827
C08462=1168.866,114.493,-53.397,-178.870,6.384,148.828
C08463=1168.871,114.245,-53.378,-178.872,6.383,148.828
C08464=1168.875,113.995,-53.359,-178.875,6.382,148.828
C08465=1168.881,113.747,-53.340,-178.878,6.380,148.829
C08466=1168.886,113.496,-53.321,-178.881,6.378,148.830
C08467=1168.890,113.248,-53.302,-178.883,6.378,148.830
C08468=1168.895,112.998,-53.282,-178.886,6.376,148.830
C08469=1168.900,112.750,-53.264,-178.889,6.374,148.831
C08470=1168.905,112.499,-53.245,-178.892,6.373,148.831
C08471=1168.909,112.251,-53.226,-178.894,6.372,148.832
C08472=1168.914,112.001,-53.206,-178.897,6.370,148.832
C08473=1168.919,111.752,-53.188,-178.899,6.368,148.833
C08474=1168.924,111.503,-53.169,-178.903,6.367,148.833
C08475=1168.928,111.254,-53.150,-178.905,6.366,148.834
C08476=1168.934,111.005,-53.131,-178.907,6.364,148.834
C08477=1168.938,110.755,-53.112,-178.910,6.363,148.834
C08478=1168.943,110.506,-53.093,-178.913,6.361,148.835
C08479=1168.948,110.257,-53.075,-178.915,6.360,148.835
C08480=1168.953,110.008,-53.055,-178.918,6.359,148.836
C08481=1168.958,109.758,-53.037,-178.921,6.357,148.837
C08482=1168.963,109.509,-53.018,-178.923,6.356,148.837
C08483=1168.967,109.260,-52.999,-178.926,6.355,148.837
C08484=1168.972,109.010,-52.980,-178.929,6.353,148.838
C08485=1168.977,108.762,-52.961,-178.932,6.352,148.838
C08486=1168.982,108.512,-52.943,-178.934,6.351,148.839
C08487=1168.986,108.263,-52.924,-178.937,6.349,148.839
C08488=1168.991,108.014,-52.906,-178.940,6.347,148.840
C08489=1168.996,107.764,-52.886,-178.942,6.347,148.840
C08490=1169.001,107.515,-52.868,-178.945,6.345,148.841
C08491=1169.006,107.266,-52.849,-178.948,6.343,148.841
C08492=1169.011,107.016,-52.831,-178.951,6.342,148.842
C08493=1169.015,106.768,-52.812,-178.953,6.341,148.842
C08494=1169.021,106.499,-52.792,-178.956,6.339,148.843
C08495=1169.026,106.230,-52.771,-178.959,6.338,148.843
C08496=1169.031,105.962,-52.751,-178.962,6.336,148.844
C08497=1169.037,105.694,-52.731,-178.965,6.335,148.844
C08498=1169.042,105.444,-52.713,-178.968,6.333,148.845
C08499=1169.046,105.195,-52.694,-178.970,6.332,148.845
C08500=1169.051,104.946,-52.676,-178.973,6.331,148.846
C08501=1169.056,104.697,-52.657,-178.976,6.329,148.846
C08502=1169.060,104.447,-52.639,-178.978,6.328,148.846
C08503=1169.066,104.198,-52.620,-178.981,6.327,148.847
C08504=1169.071,103.949,-52.601,-178.984,6.325,148.848
C08505=1169.075,103.699,-52.583,-178.986,6.324,148.848
C08506=1169.081,103.450,-52.565,-178.989,6.323,148.848
C08507=1169.085,103.201,-52.546,-178.992,6.321,148.849
C08508=1169.090,102.952,-52.528,-178.994,6.320,148.849
C08509=1169.094,102.702,-52.509,-178.997,6.319,148.850
C08510=1169.100,102.453,-52.490,-179.000,6.317,148.850
C08511=1169.105,102.204,-52.472,-179.002,6.316,148.851
C08512=1169.109,101.954,-52.454,-179.005,6.315,148.851
C08513=1169.114,101.705,-52.436,-179.008,6.313,148.852
C08514=1169.119,101.456,-52.417,-179.010,6.312,148.852
C08515=1169.124,101.207,-52.399,-179.013,6.311,148.853
C08516=1169.128,100.957,-52.380,-179.016,6.309,148.853
C08517=1169.133,100.708,-52.362,-179.018,6.308,148.854
C08518=1169.139,100.459,-52.343,-179.021,6.307,148.854
C08519=1169.144,100.210,-52.325,-179.024,6.305,148.855
C08520=1169.148,99.960,-52.307,-179.026,6.305,148.855
C08521=1169.153,99.711,-52.289,-179.029,6.303,148.856
C08522=1169.158,99.462,-52.271,-179.032,6.301,148.856
C08523=1169.163,99.213,-52.253,-179.034,6.301,148.857
C08524=1169.168,98.964,-52.233,-179.037,6.299,148.857
C08525=1169.172,98.714,-52.215,-179.040,6.298,148.858
C08526=1169.177,98.465,-52.197,-179.042,6.297,148.858
C08527=1169.182,98.216,-52.179,-179.045,6.295,148.859
C08528=1169.187,97.966,-52.161,-179.048,6.294,148.859
C08529=1169.192,97.717,-52.143,-179.050,6.293,148.860
C08530=1169.196,97.467,-52.125,-179.053,6.291,148.860
C08531=1169.202,97.218,-52.106,-179.056,6.290,148.861
C08532=1169.207,96.969,-52.088,-179.058,6.289,148.861
C08533=1169.212,96.719,-52.070,-179.061,6.287,148.862
C08534=1169.216,96.471,-52.052,-179.064,6.286,148.862
C08535=1169.221,96.222,-52.034,-179.066,6.285,148.863
C08536=1169.226,95.972,-52.015,-179.069,6.283,148.863
C08537=1169.231,95.723,-51.997,-179.072,6.282,148.864
C08538=1169.235,95.473,-51.979,-179.074,6.281,148.864
C08539=1169.240,95.224,-51.961,-179.077,6.280,148.865
C08540=1169.245,94.975,-51.943,-179.080,6.279,148.865
C08541=1169.250,94.726,-51.925,-179.083,6.277,148.866
C08542=1169.255,94.477,-51.907,-179.085,6.276,148.866
C08543=1169.260,94.226,-51.890,-179.088,6.275,148.867
C08544=1169.265,93.977,-51.871,-179.091,6.273,148.867
C08545=1169.270,93.728,-51.853,-179.093,6.272,148.867
C08546=1169.275,93.478,-51.835,-179.096,6.271,148.868
C08547=1169.280,93.229,-51.817,-179.098,6.270,148.869
C08548=1169.285,92.980,-51.799,-179.101,6.268,148.869
C08549=1169.290,92.731,-51.781,-179.104,6.267,148.870
C08550=1169.295,92.482,-51.763,-179.106,6.266,148.870
C08551=1169.300,92.233,-51.745,-179.109,6.264,148.871
C08552=1169.304,91.984,-51.728,-179.111,6.264,148.871
C08553=1169.309,91.733,-51.710,-179.114,6.262,148.872
C08554=1169.313,91.484,-51.692,-179.117,6.261,148.872
C08555=1169.318,91.235,-51.674,-179.120,6.260,148.873
C08556=1169.323,90.986,-51.656,-179.122,6.258,148.873
C08557=1169.328,90.737,-51.638,-179.125,6.257,148.874
C08558=1169.333,90.487,-51.620,-179.128,6.256,148.874
C08559=1169.338,90.238,-51.603,-179.130,6.254,148.874
C08560=1169.343,89.988,-51.585,-179.133,6.253,148.875
C08561=1169.348,89.739,-51.567,-179.136,6.252,148.876
C08562=1169.353,89.490,-51.549,-179.138,6.251,148.876
C08563=1169.358,89.241,-51.531,-179.141,6.250,148.877
C08564=1169.363,88.991,-51.514,-179.143,6.249,148.877
C08565=1169.367,88.742,-51.497,-179.146,6.247,148.878
C08566=1169.372,88.493,-51.479,-179.149,6.246,148.878
C08567=1169.377,88.243,-51.461,-179.151,6.245,148.879
C08568=1169.382,87.994,-51.443,-179.154,6.243,148.879
C08569=1169.387,87.745,-51.425,-179.157,6.242,148.880
C08570=1169.392,87.496,-51.407,-179.160,6.241,148.880
C08571=1169.397,87.246,-51.390,-179.163,6.239,148.881
C08572=1169.402,86.997,-51.372,-179.165,6.239,148.881
C08573=1169.407,86.748,-51.355,-179.168,6.237,148.882
C08574=1169.412,86.498,-51.338,-179.170,6.236,148.882
C08575=1169.417,86.249,-51.320,-179.173,6.235,148.883
C08576=1169.422,85.999,-51.302,-179.175,6.234,148.883
C08577=1169.427,85.750,-51.284,-179.178,6.232,148.884
C08578=1169.431,85.501,-51.267,-179.181,6.232,148.884
C08579=1169.436,85.251,-51.250,-179.183,6.230,148.885
C08580=1169.441,85.002,-51.232,-179.186,6.228,148.885
C08581=1169.446,84.752,-51.214,-179.189,6.228,148.886
C08582=1169.450,84.503,-51.197,-179.192,6.226,148.886
C08583=1169.455,84.254,-51.179,-179.194,6.226,148.887
C08584=1169.461,84.004,-51.162,-179.197,6.224,148.887
C08585=1169.466,83.755,-51.144,-179.199,6.223,148.888
C08586=1169.470,83.506,-51.127,-179.202,6.222,148.888
C08587=1169.475,83.257,-51.109,-179.204,6.221,148.889
C08588=1169.480,83.007,-51.092,-179.208,6.220,148.889
C08589=1169.485,82.758,-51.074,-179.210,6.219,148.890
C08590=1169.490,82.509,-51.058,-179.213,6.217,148.891
C08591=1169.495,82.260,-51.040,-179.216,6.216,148.891
C08592=1169.500,82.010,-51.022,-179.218,6.215,148.891
C08593=1169.504,81.761,-51.005,-179.221,6.213,148.892
C08594=1169.510,81.511,-50.988,-179.223,6.212,148.892
C08595=1169.515,81.262,-50.970,-179.226,6.211,148.893
C08596=1169.520,81.012,-50.952,-179.229,6.210,148.894
C08597=1169.524,80.763,-50.936,-179.231,6.209,148.894
C08598=1169.530,80.495,-50.917,-179.234,6.208,148.895
C08599=1169.535,80.226,-50.898,-179.237,6.207,148.895
C08600=1169.540,79.958,-50.880,-179.240,6.205,148.896
C08601=1169.545,79.689,-50.861,-179.243,6.204,148.896
C08602=1169.551,79.440,-50.844,-179.245,6.203,148.897
C08603=1169.555,79.191,-50.827,-179.248,6.201,148.897
C08604=1169.560,78.942,-50.809,-179.251,6.201,148.898
C08605=1169.565,78.692,-50.792,-179.253,6.199,148.898
C08606=1169.570,78.442,-50.775,-179.256,6.198,148.899
C08607=1169.575,78.193,-50.757,-179.259,6.197,148.899
C08608=1169.580,77.945,-50.741,-179.261,6.196,148.900
C08609=1169.585,77.695,-50.724,-179.264,6.194,148.900
C08610=1169.590,77.445,-50.706,-179.267,6.194,148.901
C08611=1169.595,77.196,-50.689,-179.269,6.192,148.902
C08612=1169.600,76.946,-50.672,-179.271,6.191,148.902
C08613=1169.604,76.697,-50.655,-179.275,6.190,148.903
C08614=1169.610,76.448,-50.637,-179.277,6.189,148.903
C08615=1169.614,76.199,-50.621,-179.280,6.188,148.904
C08616=1169.619,75.949,-50.603,-179.282,6.187,148.904
C08617=1169.624,75.700,-50.587,-179.285,6.186,148.905
C08618=1169.629,75.450,-50.569,-179.288,6.185,148.905
C08619=1169.634,75.202,-50.552,-179.290,6.183,148.906
C08620=1169.639,74.952,-50.535,-179.293,6.182,148.906
C08621=1169.644,74.702,-50.519,-179.296,6.181,148.907
C08622=1169.649,74.453,-50.501,-179.298,6.180,148.907
C08623=1169.654,74.204,-50.485,-179.301,6.179,148.908
C08624=1169.659,73.955,-50.467,-179.304,6.178,148.908
C08625=1169.663,73.705,-50.450,-179.306,6.176,148.909
C08626=1169.669,73.455,-50.433,-179.309,6.176,148.910
C08627=1169.673,73.206,-50.416,-179.312,6.174,148.910
C08628=1169.679,72.957,-50.399,-179.314,6.173,148.910
C08629=1169.683,72.707,-50.383,-179.316,6.173,148.911
C08630=1169.689,72.457,-50.366,-179.319,6.171,148.911
C08631=1169.693,72.208,-50.349,-179.322,6.171,148.912
C08632=1169.699,71.959,-50.332,-179.325,6.169,148.913
C08633=1169.703,71.709,-50.315,-179.327,6.168,148.913
C08634=1169.708,71.461,-50.298,-179.330,6.167,148.914
C08635=1169.713,71.211,-50.281,-179.333,6.166,148.914
C08636=1169.718,70.962,-50.264,-179.335,6.164,148.915
C08637=1169.723,70.712,-50.247,-179.338,6.164,148.915
C08638=1169.727,70.463,-50.230,-179.341,6.162,148.916
C08639=1169.733,70.214,-50.214,-179.343,6.161,148.916
C08640=1169.738,69.964,-50.197,-179.346,6.160,148.917
C08641=1169.742,69.715,-50.180,-179.348,6.159,148.917
C08642=1169.747,69.466,-50.164,-179.351,6.159,148.918
C08643=1169.753,69.216,-50.147,-179.354,6.157,148.918
C08644=1169.757,68.967,-50.130,-179.356,6.156,148.919
C08645=1169.762,68.718,-50.114,-179.359,6.155,148.920
C08646=1169.767,68.468,-50.096,-179.362,6.154,148.920
C08647=1169.772,68.218,-50.080,-179.364,6.153,148.921
C08648=1169.777,67.969,-50.064,-179.367,6.152,148.921
C08649=1169.782,67.719,-50.047,-179.370,6.150,148.922
C08650=1169.787,67.470,-50.030,-179.372,6.150,148.922
C08651=1169.792,67.221,-50.014,-179.374,6.149,148.923
C08652=1169.797,66.971,-49.997,-179.377,6.147,148.923
C08653=1169.802,66.722,-49.980,-179.380,6.147,148.924
C08654=1169.807,66.473,-49.964,-179.383,6.145,148.924
C08655=1169.811,66.223,-49.947,-179.385,6.145,148.925
C08656=1169.817,65.973,-49.930,-179.388,6.143,148.925
C08657=1169.822,65.724,-49.914,-179.391,6.142,148.926
C08658=1169.826,65.475,-49.897,-179.393,6.141,148.927
C08659=1169.832,65.226,-49.881,-179.396,6.140,148.927
C08660=1169.837,64.976,-49.864,-179.398,6.139,148.928
C08661=1169.841,64.727,-49.847,-179.401,6.138,148.928
C08662=1169.847,64.477,-49.832,-179.403,6.137,148.929
C08663=1169.851,64.228,-49.815,-179.407,6.136,148.929
C08664=1169.857,63.979,-49.798,-179.409,6.135,148.930
C08665=1169.861,63.729,-49.781,-179.411,6.134,148.930
C08666=1169.866,63.479,-49.765,-179.414,6.133,148.931
C08667=1169.871,63.230,-49.749,-179.417,6.132,148.932
C08668=1169.876,62.981,-49.732,-179.420,6.130,148.932
C08669=1169.881,62.732,-49.716,-179.422,6.130,148.933
C08670=1169.886,62.482,-49.700,-179.424,6.129,148.933
C08671=1169.891,62.233,-49.683,-179.428,6.128,148.934
C08672=1169.896,61.983,-49.667,-179.430,6.127,148.934
C08673=1169.901,61.733,-49.651,-179.433,6.126,148.935
C08674=1169.906,61.485,-49.634,-179.435,6.125,148.935
C08675=1169.911,61.235,-49.617,-179.438,6.124,148.936
C08676=1169.916,60.985,-49.602,-179.440,6.123,148.936
C08677=1169.921,60.736,-49.585,-179.443,6.122,148.937
C08678=1169.926,60.487,-49.569,-179.446,6.120,148.937
C08679=1169.931,60.237,-49.553,-179.448,6.120,148.938
C08680=1169.936,59.988,-49.536,-179.451,6.119,148.939
C08681=1169.940,59.739,-49.520,-179.453,6.117,148.939
C08682=1169.946,59.489,-49.504,-179.456,6.117,148.940
C08683=1169.951,59.239,-49.487,-179.459,6.115,148.940
C08684=1169.956,58.990,-49.471,-179.461,6.115,148.941
C08685=1169.961,58.741,-49.455,-179.463,6.114,148.941
C08686=1169.966,58.492,-49.438,-179.467,6.112,148.942
C08687=1169.971,58.242,-49.422,-179.469,6.112,148.942
C08688=1169.976,57.993,-49.406,-179.472,6.110,148.943
C08689=1169.980,57.743,-49.390,-179.474,6.109,148.943
C08690=1169.985,57.494,-49.374,-179.477,6.109,148.944
C08691=1169.990,57.244,-49.358,-179.480,6.107,148.945
C08692=1169.995,56.995,-49.341,-179.482,6.107,148.945
C08693=1170.000,56.745,-49.325,-179.485,6.106,148.946
C08694=1170.005,56.496,-49.309,-179.488,6.104,148.946
C08695=1170.010,56.246,-49.293,-179.490,6.104,148.947
C08696=1170.015,55.997,-49.277,-179.493,6.102,148.947
C08697=1170.020,55.747,-49.261,-179.496,6.102,148.948
C08698=1170.025,55.499,-49.245,-179.498,6.101,148.949
C08699=1170.030,55.249,-49.229,-179.501,6.100,148.949
C08700=1170.035,54.999,-49.213,-179.503,6.099,148.950
C08701=1170.040,54.750,-49.197,-179.506,6.098,148.950
C08702=1170.045,54.481,-49.179,-179.509,6.097,148.951
C08703=1170.051,54.213,-49.162,-179.511,6.096,148.951
C08704=1170.056,53.944,-49.145,-179.514,6.095,148.952
C08705=1170.062,53.676,-49.128,-179.517,6.094,148.952
C08706=1170.066,53.426,-49.112,-179.520,6.093,148.953
C08707=1170.072,53.177,-49.096,-179.522,6.092,148.954
C08708=1170.076,52.927,-49.079,-179.525,6.091,148.954
C08709=1170.082,52.678,-49.064,-179.527,6.089,148.955
C08710=1170.087,52.428,-49.048,-179.530,6.089,148.955
C08711=1170.091,52.179,-49.032,-179.533,6.088,148.956
C08712=1170.097,51.930,-49.016,-179.535,6.087,148.956
C08713=1170.102,51.680,-49.000,-179.538,6.086,148.957
C08714=1170.106,51.431,-48.984,-179.541,6.085,148.958
C08715=1170.111,51.182,-48.969,-179.543,6.084,148.958
C08716=1170.116,50.931,-48.953,-179.545,6.083,148.959
C08717=1170.121,50.682,-48.937,-179.549,6.082,148.959
C08718=1170.127,50.433,-48.921,-179.551,6.081,148.960
C08719=1170.131,50.183,-48.905,-179.553,6.081,148.960
C08720=1170.137,49.934,-48.889,-179.556,6.079,148.961
C08721=1170.141,49.685,-48.874,-179.559,6.078,148.962
C08722=1170.146,49.435,-48.858,-179.561,6.078,148.962
C08723=1170.151,49.186,-48.842,-179.564,6.076,148.963
C08724=1170.157,48.936,-48.827,-179.566,6.075,148.963
C08725=1170.161,48.686,-48.811,-179.569,6.075,148.964
C08726=1170.167,48.437,-48.794,-179.571,6.074,148.964
C08727=1170.171,48.188,-48.779,-179.574,6.073,148.965
C08728=1170.176,47.938,-48.763,-179.577,6.072,148.965
C08729=1170.181,47.689,-48.748,-179.579,6.071,148.966
C08730=1170.187,47.439,-48.732,-179.582,6.070,148.967
C08731=1170.192,47.189,-48.716,-179.585,6.069,148.967
C08732=1170.196,46.941,-48.701,-179.587,6.069,148.968
C08733=1170.201,46.692,-48.685,-179.590,6.067,148.968
C08734=1170.206,46.441,-48.669,-179.593,6.066,148.969
C08735=1170.211,46.192,-48.653,-179.595,6.066,148.969
C08736=1170.216,45.943,-48.638,-179.598,6.064,148.970
C08737=1170.221,45.694,-48.623,-179.600,6.063,148.970
C08738=1170.226,45.443,-48.607,-179.603,6.063,148.971
C08739=1170.232,45.194,-48.591,-179.605,6.062,148.972
C08740=1170.236,44.945,-48.576,-179.608,6.061,148.972
C08741=1170.241,44.695,-48.560,-179.611,6.060,148.973
C08742=1170.246,44.445,-48.545,-179.613,6.059,148.973
C08743=1170.251,44.196,-48.530,-179.616,6.058,148.974
C08744=1170.256,43.947,-48.514,-179.618,6.057,148.974
C08745=1170.261,43.697,-48.498,-179.621,6.057,148.975
C08746=1170.266,43.448,-48.483,-179.624,6.055,148.976
C08747=1170.271,43.198,-48.468,-179.626,6.055,148.976
C08748=1170.277,42.949,-48.452,-179.629,6.054,148.977
C08749=1170.281,42.699,-48.437,-179.631,6.053,148.977
C08750=1170.286,42.450,-48.421,-179.634,6.052,148.978
C08751=1170.292,42.200,-48.405,-179.637,6.051,148.979
C08752=1170.296,41.951,-48.390,-179.639,6.051,148.979
C08753=1170.302,41.702,-48.375,-179.641,6.050,148.980
C08754=1170.306,41.452,-48.359,-179.645,6.048,148.980
C08755=1170.311,41.203,-48.344,-179.647,6.048,148.981
C08756=1170.316,40.953,-48.328,-179.649,6.047,148.981
C08757=1170.322,40.704,-48.313,-179.652,6.045,148.982
C08758=1170.326,40.455,-48.298,-179.655,6.045,148.983
C08759=1170.331,40.205,-48.282,-179.657,6.044,148.983
C08760=1170.336,39.956,-48.267,-179.660,6.044,148.984
C08761=1170.341,39.706,-48.251,-179.663,6.042,148.984
C08762=1170.347,39.456,-48.236,-179.665,6.041,148.985
C08763=1170.352,39.207,-48.221,-179.668,6.041,148.985
C08764=1170.357,38.958,-48.206,-179.670,6.040,148.986
C08765=1170.361,38.708,-48.190,-179.673,6.039,148.987
C08766=1170.366,38.458,-48.175,-179.675,6.038,148.987
C08767=1170.371,38.209,-48.160,-179.678,6.037,148.988
C08768=1170.377,37.959,-48.145,-179.680,6.037,148.988
C08769=1170.382,37.710,-48.129,-179.683,6.035,148.989
C08770=1170.387,37.461,-48.114,-179.686,6.035,148.989
C08771=1170.392,37.211,-48.099,-179.688,6.034,148.990
C08772=1170.396,36.962,-48.083,-179.691,6.033,148.991
C08773=1170.402,36.712,-48.069,-179.693,6.032,148.991
C08774=1170.407,36.463,-48.054,-179.696,6.031,148.992
C08775=1170.412,36.213,-48.038,-179.698,6.030,148.992
C08776=1170.417,35.964,-48.023,-179.701,6.030,148.993
C08777=1170.422,35.714,-48.008,-179.704,6.028,148.993
C08778=1170.427,35.465,-47.993,-179.706,6.028,148.994
C08779=1170.432,35.216,-47.978,-179.709,6.027,148.995
C08780=1170.437,34.966,-47.963,-179.711,6.026,148.995
C08781=1170.442,34.716,-47.947,-179.714,6.025,148.996
C08782=1170.447,34.467,-47.932,-179.716,6.024,148.996
C08783=1170.452,34.217,-47.917,-179.719,6.024,148.997
C08784=1170.457,33.967,-47.902,-179.721,6.023,148.997
C08785=1170.462,33.718,-47.887,-179.724,6.022,148.998
C08786=1170.467,33.468,-47.873,-179.727,6.021,148.999
C08787=1170.472,33.219,-47.858,-179.729,6.020,148.999
C08788=1170.477,32.970,-47.842,-179.732,6.020,149.000
C08789=1170.482,32.720,-47.828,-179.734,6.019,149.000
C08790=1170.488,32.471,-47.812,-179.737,6.018,149.001
C08791=1170.492,32.222,-47.797,-179.739,6.017,149.001
C08792=1170.497,31.972,-47.783,-179.742,6.016,149.002
C08793=1170.503,31.723,-47.767,-179.745,6.016,149.003
C08794=1170.508,31.473,-47.753,-179.748,6.014,149.003
C08795=1170.512,31.223,-47.738,-179.750,6.014,149.004
C08796=1170.517,30.973,-47.723,-179.752,6.013,149.004
C08797=1170.522,30.724,-47.708,-179.755,6.012,149.005
C08798=1170.527,30.475,-47.692,-179.758,6.012,149.006
C08799=1170.532,30.225,-47.678,-179.760,6.010,149.006
C08800=1170.537,29.976,-47.663,-179.763,6.010,149.007
C08801=1170.543,29.726,-47.648,-179.765,6.009,149.007
C08802=1170.547,29.477,-47.633,-179.768,6.008,149.008
C08803=1170.552,29.227,-47.619,-179.770,6.008,149.008
C08804=1170.558,28.978,-47.603,-179.773,6.006,149.009
C08805=1170.563,28.728,-47.589,-179.776,6.006,149.010
C08806=1170.568,28.459,-47.573,-179.778,6.005,149.010
C08807=1170.574,28.190,-47.557,-179.781,6.004,149.011
C08808=1170.579,27.921,-47.541,-179.784,6.003,149.012
C08809=1170.585,27.653,-47.526,-179.787,6.003,149.012
C08810=1170.590,27.404,-47.510,-179.789,6.002,149.013
C08811=1170.595,27.154,-47.496,-179.792,6.001,149.013
C08812=1170.600,26.904,-47.482,-179.794,6.000,149.014
C08813=1170.605,26.655,-47.466,-179.797,5.999,149.014
C08814=1170.610,26.405,-47.452,-179.799,5.999,149.015
C08815=1170.615,26.156,-47.437,-179.802,5.998,149.016
C08816=1170.620,25.906,-47.423,-179.805,5.997,149.016
C08817=1170.626,25.656,-47.408,-179.807,5.996,149.017
C08818=1170.630,25.407,-47.393,-179.810,5.995,149.017
C08819=1170.635,25.157,-47.378,-179.812,5.995,149.018
C08820=1170.640,24.908,-47.364,-179.814,5.994,149.019
C08821=1170.645,24.659,-47.349,-179.817,5.993,149.019
C08822=1170.650,24.409,-47.334,-179.820,5.992,149.020
C08823=1170.655,24.159,-47.320,-179.822,5.991,149.020
C08824=1170.660,23.910,-47.305,-179.825,5.991,149.021
C08825=1170.665,23.660,-47.291,-179.827,5.990,149.021
C08826=1170.670,23.410,-47.277,-179.830,5.989,149.022
C08827=1170.676,23.162,-47.261,-179.832,5.989,149.023
C08828=1170.681,22.912,-47.247,-179.835,5.987,149.023
C08829=1170.686,22.662,-47.233,-179.838,5.987,149.024
C08830=1170.691,22.413,-47.218,-179.840,5.986,149.024
C08831=1170.695,22.164,-47.203,-179.843,5.986,149.025
C08832=1170.700,21.914,-47.189,-179.845,5.985,149.026
C08833=1170.705,21.664,-47.175,-179.848,5.984,149.026
C08834=1170.711,21.414,-47.160,-179.850,5.983,149.027
C08835=1170.716,21.165,-47.145,-179.853,5.982,149.027
C08836=1170.721,20.916,-47.131,-179.856,5.982,149.028
C08837=1170.726,20.666,-47.117,-179.858,5.981,149.029
C08838=1170.731,20.417,-47.103,-179.860,5.980,149.029
C08839=1170.736,20.167,-47.088,-179.863,5.979,149.030
C08840=1170.741,19.918,-47.073,-179.866,5.978,149.030
C08841=1170.746,19.668,-47.059,-179.869,5.978,149.031
C08842=1170.751,19.418,-47.045,-179.871,5.977,149.031
C08843=1170.757,19.169,-47.030,-179.873,5.976,149.032
C08844=1170.762,18.919,-47.016,-179.875,5.976,149.033
C08845=1170.767,18.670,-47.002,-179.878,5.975,149.033
C08846=1170.772,18.420,-46.987,-179.881,5.975,149.034
C08847=1170.777,18.170,-46.973,-179.884,5.973,149.034
C08848=1170.781,17.921,-46.958,-179.886,5.972,149.035
C08849=1170.787,17.672,-46.944,-179.888,5.972,149.036
C08850=1170.792,17.422,-46.930,-179.891,5.971,149.036
C08851=1170.797,17.173,-46.916,-179.894,5.971,149.037
C08852=1170.802,16.923,-46.901,-179.896,5.970,149.037
C08853=1170.807,16.673,-46.887,-179.898,5.969,149.038
C08854=1170.812,16.424,-46.873,-179.901,5.969,149.039
C08855=1170.817,16.174,-46.859,-179.904,5.967,149.039
C08856=1170.822,15.925,-46.845,-179.907,5.967,149.040
C08857=1170.827,15.675,-46.830,-179.909,5.966,149.040
C08858=1170.832,15.425,-46.816,-179.911,5.965,149.041
C08859=1170.838,15.176,-46.802,-179.914,5.965,149.042
C08860=1170.843,14.927,-46.788,-179.916,5.964,149.042
C08861=1170.848,14.677,-46.774,-179.919,5.964,149.043
C08862=1170.853,14.427,-46.759,-179.921,5.963,149.043
C08863=1170.858,14.178,-46.745,-179.924,5.962,149.044
C08864=1170.863,13.929,-46.731,-179.927,5.961,149.045
C08865=1170.868,13.679,-46.717,-179.929,5.960,149.045
C08866=1170.873,13.429,-46.703,-179.932,5.960,149.046
C08867=1170.879,13.180,-46.689,-179.934,5.959,149.046
C08868=1170.884,12.930,-46.674,-179.936,5.958,149.047
C08869=1170.888,12.681,-46.660,-179.939,5.958,149.048
C08870=1170.893,12.431,-46.646,-179.941,5.957,149.048
C08871=1170.898,12.182,-46.633,-179.944,5.957,149.049
C08872=1170.903,11.932,-46.619,-179.946,5.956,149.049
C08873=1170.908,11.682,-46.605,-179.949,5.955,149.050
C08874=1170.913,11.432,-46.590,-179.952,5.954,149.051
C08875=1170.919,11.183,-46.577,-179.954,5.953,149.051
C08876=1170.924,10.934,-46.562,-179.957,5.953,149.052
C08877=1170.929,10.684,-46.548,-179.959,5.952,149.052
C08878=1170.934,10.435,-46.534,-179.962,5.951,149.053
C08879=1170.939,10.186,-46.520,-179.964,5.951,149.054
C08880=1170.944,9.935,-46.507,-179.966,5.950,149.054
C08881=1170.949,9.686,-46.493,-179.969,5.950,149.055
C08882=1170.954,9.437,-46.479,-179.972,5.949,149.055
C08883=1170.959,9.187,-46.464,-179.974,5.948,149.056
C08884=1170.964,8.937,-46.450,-179.977,5.947,149.057
C08885=1170.970,8.688,-46.437,-179.979,5.946,149.057
C08886=1170.974,8.438,-46.423,-179.982,5.946,149.058
C08887=1170.979,8.188,-46.409,-179.985,5.945,149.058
C08888=1170.985,7.939,-46.395,-179.987,5.944,149.059
C08889=1170.990,7.689,-46.381,-179.989,5.944,149.060
C08890=1170.995,7.439,-46.367,-179.992,5.943,149.060
C08891=1171.000,7.191,-46.354,-179.994,5.943,149.061
C08892=1171.005,6.941,-46.340,-179.997,5.942,149.061
C08893=1171.011,6.691,-46.326,-179.999,5.941,149.062
C08894=1171.016,6.442,-46.312,179.998,5.941,149.063
C08895=1171.020,6.192,-46.298,179.996,5.940,149.063
C08896=1171.026,5.943,-46.285,179.993,5.940,149.064
C08897=1171.031,5.693,-46.271,179.990,5.938,149.064
C08898=1171.036,5.443,-46.257,179.988,5.938,149.065
C08899=1171.041,5.194,-46.244,179.985,5.937,149.065
C08900=1171.046,4.944,-46.230,179.983,5.937,149.066
C08901=1171.051,4.695,-46.216,179.981,5.936,149.067
C08902=1171.057,4.445,-46.202,179.978,5.935,149.067
C08903=1171.061,4.195,-46.189,179.975,5.935,149.068
C08904=1171.066,3.946,-46.175,179.973,5.934,149.068
C08905=1171.072,3.696,-46.161,179.970,5.934,149.069
C08906=1171.076,3.447,-46.148,179.968,5.933,149.070
C08907=1171.081,3.198,-46.134,179.966,5.932,149.070
C08908=1171.087,2.947,-46.120,179.963,5.932,149.071
C08909=1171.092,2.698,-46.106,179.961,5.931,149.071
C08910=1171.097,2.429,-46.092,179.958,5.930,149.072
C08911=1171.103,2.159,-46.077,179.955,5.929,149.073
C08912=1171.108,1.890,-46.062,179.952,5.929,149.074
C08913=1171.114,1.621,-46.048,179.950,5.928,149.074
C08914=1171.119,1.371,-46.034,179.947,5.927,149.075
C08915=1171.124,1.122,-46.021,179.945,5.927,149.075
C08916=1171.129,0.872,-46.007,179.943,5.926,149.076
C08917=1171.134,0.623,-45.994,179.940,5.926,149.077
C08918=1171.139,0.373,-45.980,179.937,5.925,149.077
C08919=1171.145,0.123,-45.966,179.935,5.924,149.078
C08920=1171.149,-0.126,-45.953,179.932,5.924,149.078
C08921=1171.155,-0.376,-45.939,179.930,5.923,149.079
C08922=1171.160,-0.625,-45.925,179.928,5.923,149.080
C08923=1171.165,-0.875,-45.912,179.925,5.922,149.080
C08924=1171.170,-1.124,-45.899,179.923,5.921,149.081
C08925=1171.175,-1.374,-45.886,179.920,5.921,149.081
C08926=1171.181,-1.624,-45.872,179.917,5.920,149.082
C08927=1171.185,-1.873,-45.859,179.915,5.920,149.082
C08928=1171.191,-2.123,-45.846,179.912,5.918,149.083
C08929=1171.196,-2.372,-45.831,179.909,5.918,149.084
C08930=1171.201,-2.622,-45.819,179.907,5.917,149.084
C08931=1171.206,-2.872,-45.804,179.905,5.917,149.085
C08932=1171.211,-3.121,-45.792,179.902,5.916,149.085
C08933=1171.216,-3.371,-45.778,179.900,5.915,149.086
C08934=1171.221,-3.620,-45.765,179.897,5.915,149.087
C08935=1171.226,-3.870,-45.751,179.895,5.914,149.087
C08936=1171.231,-4.119,-45.739,179.892,5.914,149.088
C08937=1171.236,-4.369,-45.724,179.890,5.913,149.089
C08938=1171.241,-4.619,-45.712,179.887,5.912,149.089
C08939=1171.247,-4.868,-45.699,179.885,5.912,149.090
C08940=1171.251,-5.118,-45.685,179.883,5.911,149.090
C08941=1171.257,-5.367,-45.672,179.880,5.911,149.091
C08942=1171.262,-5.617,-45.659,179.877,5.910,149.092
C08943=1171.267,-5.866,-45.645,179.875,5.909,149.092
C08944=1171.272,-6.116,-45.632,179.872,5.909,149.093
C08945=1171.278,-6.366,-45.619,179.870,5.908,149.094
C08946=1171.282,-6.615,-45.605,179.868,5.907,149.094
C08947=1171.288,-6.865,-45.592,179.865,5.907,149.095
C08948=1171.293,-7.114,-45.579,179.863,5.906,149.095
C08949=1171.298,-7.365,-45.566,179.860,5.906,149.096
C08950=1171.303,-7.613,-45.552,179.857,5.905,149.097
C08951=1171.308,-7.864,-45.539,179.855,5.904,149.097
C08952=1171.313,-8.113,-45.526,179.853,5.904,149.098
C08953=1171.318,-8.363,-45.513,179.850,5.904,149.098
C08954=1171.324,-8.613,-45.500,179.848,5.903,149.099
C08955=1171.329,-8.861,-45.487,179.845,5.902,149.100
C08956=1171.334,-9.112,-45.473,179.843,5.901,149.100
C08957=1171.339,-9.361,-45.461,179.840,5.901,149.101
C08958=1171.344,-9.611,-45.448,179.838,5.901,149.101
C08959=1171.349,-9.861,-45.434,179.835,5.900,149.102
C08960=1171.354,-10.109,-45.421,179.833,5.899,149.103
C08961=1171.359,-10.360,-45.408,179.831,5.900,149.103
C08962=1171.365,-10.609,-45.395,179.829,5.899,149.104
C08963=1171.370,-10.858,-45.382,179.826,5.898,149.104
C08964=1171.375,-11.109,-45.369,179.823,5.898,149.105
C08965=1171.380,-11.358,-45.356,179.821,5.897,149.106
C08966=1171.385,-11.608,-45.343,179.818,5.897,149.106
C08967=1171.391,-11.857,-45.330,179.816,5.896,149.107
C08968=1171.395,-12.106,-45.317,179.814,5.895,149.107
C08969=1171.400,-12.356,-45.304,179.811,5.895,149.108
C08970=1171.406,-12.606,-45.291,179.809,5.894,149.109
C08971=1171.411,-12.855,-45.278,179.806,5.894,149.109
C08972=1171.415,-13.105,-45.265,179.803,5.893,149.110
C08973=1171.421,-13.355,-45.252,179.801,5.892,149.110
C08974=1171.426,-13.604,-45.239,179.799,5.892,149.111
C08975=1171.431,-13.854,-45.226,179.796,5.891,149.112
C08976=1171.437,-14.104,-45.213,179.794,5.891,149.112
C08977=1171.442,-14.353,-45.200,179.791,5.890,149.113
C08978=1171.446,-14.603,-45.187,179.789,5.889,149.113
C08979=1171.451,-14.852,-45.175,179.786,5.889,149.114
C08980=1171.457,-15.102,-45.162,179.784,5.888,149.115
C08981=1171.462,-15.352,-45.149,179.781,5.888,149.115
C08982=1171.467,-15.601,-45.136,179.779,5.887,149.116
C08983=1171.472,-15.851,-45.123,179.776,5.887,149.117
C08984=1171.478,-16.100,-45.110,179.774,5.886,149.117
C08985=1171.483,-16.350,-45.097,179.771,5.885,149.118
C08986=1171.488,-16.600,-45.085,179.769,5.885,149.118
C08987=1171.493,-16.849,-45.072,179.767,5.885,149.119
C08988=1171.498,-17.099,-45.059,179.764,5.885,149.120
C08989=1171.503,-17.349,-45.046,179.762,5.884,149.120
C08990=1171.508,-17.598,-45.033,179.760,5.883,149.121
C08991=1171.513,-17.847,-45.021,179.757,5.883,149.122
C08992=1171.518,-18.098,-45.008,179.755,5.882,149.122
C08993=1171.524,-18.348,-44.995,179.752,5.882,149.123
C08994=1171.529,-18.597,-44.983,179.750,5.881,149.123
C08995=1171.534,-18.846,-44.970,179.747,5.880,149.124
C08996=1171.539,-19.096,-44.957,179.745,5.880,149.125
C08997=1171.544,-19.345,-44.945,179.742,5.879,149.125
C08998=1171.550,-19.595,-44.931,179.740,5.879,149.126
C08999=1171.555,-19.844,-44.919,179.737,5.878,149.126
C09000=1171.560,-20.094,-44.907,179.735,5.877,149.127
C09001=1171.565,-20.344,-44.894,179.732,5.877,149.128
C09002=1171.570,-20.594,-44.881,179.731,5.877,149.128
C09003=1171.575,-20.843,-44.869,179.728,5.876,149.129
C09004=1171.581,-21.093,-44.855,179.725,5.876,149.129
C09005=1171.586,-21.343,-44.843,179.723,5.875,149.130
C09006=1171.591,-21.593,-44.831,179.720,5.875,149.131
C09007=1171.596,-21.842,-44.818,179.718,5.874,149.131
C09008=1171.601,-22.091,-44.805,179.716,5.873,149.132
C09009=1171.606,-22.341,-44.793,179.713,5.873,149.132
C09010=1171.612,-22.590,-44.781,179.710,5.873,149.133
C09011=1171.616,-22.841,-44.768,179.708,5.872,149.134
C09012=1171.621,-23.090,-44.755,179.705,5.871,149.134
C09013=1171.627,-23.339,-44.742,179.703,5.870,149.135
C09014=1171.633,-23.610,-44.729,179.701,5.870,149.136
C09015=1171.638,-23.879,-44.716,179.698,5.870,149.136
C09016=1171.644,-24.149,-44.702,179.695,5.869,149.137
C09017=1171.649,-24.419,-44.689,179.693,5.869,149.138
C09018=1171.654,-24.669,-44.676,179.690,5.868,149.138
C09019=1171.659,-24.918,-44.663,179.688,5.867,149.139
C09020=1171.665,-25.168,-44.652,179.686,5.868,149.139
C09021=1171.670,-25.417,-44.639,179.684,5.867,149.140
C09022=1171.675,-25.666,-44.626,179.681,5.867,149.141
C09023=1171.680,-25.917,-44.614,179.678,5.866,149.141
C09024=1171.685,-26.166,-44.602,179.676,5.865,149.142
C09025=1171.690,-26.416,-44.589,179.673,5.865,149.142
C09026=1171.696,-26.666,-44.577,179.671,5.864,149.143
C09027=1171.701,-26.915,-44.564,179.669,5.864,149.144
C09028=1171.706,-27.165,-44.553,179.666,5.863,149.144
C09029=1171.711,-27.414,-44.540,179.664,5.862,149.145
C09030=1171.716,-27.664,-44.527,179.662,5.863,149.146
C09031=1171.721,-27.914,-44.515,179.659,5.862,149.146
C09032=1171.726,-28.163,-44.502,179.657,5.861,149.147
C09033=1171.732,-28.413,-44.491,179.654,5.861,149.147
C09034=1171.737,-28.663,-44.478,179.652,5.860,149.148
C09035=1171.742,-28.912,-44.465,179.649,5.860,149.149
C09036=1171.748,-29.162,-44.454,179.647,5.859,149.149
C09037=1171.753,-29.411,-44.441,179.644,5.858,149.150
C09038=1171.758,-29.661,-44.429,179.642,5.859,149.150
C09039=1171.763,-29.911,-44.416,179.640,5.858,149.151
C09040=1171.769,-30.161,-44.405,179.638,5.858,149.152
C09041=1171.774,-30.410,-44.392,179.635,5.857,149.152
C09042=1171.779,-30.660,-44.380,179.633,5.856,149.153
C09043=1171.783,-30.909,-44.368,179.630,5.856,149.153
C09044=1171.788,-31.159,-44.356,179.627,5.855,149.154
C09045=1171.794,-31.409,-44.343,179.625,5.855,149.155
C09046=1171.799,-31.659,-44.331,179.623,5.855,149.155
C09047=1171.804,-31.908,-44.319,179.620,5.855,149.156
C09048=1171.810,-32.158,-44.307,179.618,5.854,149.157
C09049=1171.815,-32.407,-44.294,179.616,5.853,149.157
C09050=1171.820,-32.657,-44.282,179.613,5.853,149.158
C09051=1171.826,-32.907,-44.270,179.611,5.852,149.158
C09052=1171.830,-33.156,-44.258,179.608,5.852,149.159
C09053=1171.835,-33.406,-44.247,179.606,5.851,149.160
C09054=1171.840,-33.655,-44.234,179.604,5.851,149.160
C09055=1171.846,-33.905,-44.222,179.601,5.851,149.161
C09056=1171.851,-34.155,-44.209,179.599,5.850,149.161
C09057=1171.856,-34.405,-44.198,179.596,5.850,149.162
C09058=1171.861,-34.654,-44.186,179.594,5.849,149.163
C09059=1171.866,-34.903,-44.174,179.592,5.848,149.163
C09060=1171.872,-35.153,-44.162,179.589,5.848,149.164
C09061=1171.877,-35.403,-44.150,179.587,5.848,149.164
C09062=1171.882,-35.653,-44.137,179.585,5.847,149.165
C09063=1171.888,-35.903,-44.125,179.582,5.847,149.166
C09064=1171.892,-36.152,-44.114,179.580,5.846,149.166
C09065=1171.897,-36.402,-44.102,179.577,5.846,149.167
C09066=1171.903,-36.652,-44.090,179.575,5.845,149.167
C09067=1171.908,-36.901,-44.078,179.573,5.845,149.168
C09068=1171.913,-37.151,-44.065,179.570,5.845,149.169
C09069=1171.918,-37.400,-44.054,179.568,5.844,149.169
C09070=1171.924,-37.650,-44.042,179.565,5.844,149.170
C09071=1171.929,-37.900,-44.029,179.563,5.843,149.171
C09072=1171.934,-38.150,-44.018,179.561,5.842,149.171
C09073=1171.939,-38.399,-44.006,179.558,5.843,149.172
C09074=1171.944,-38.649,-43.994,179.556,5.842,149.172
C09075=1171.949,-38.898,-43.982,179.554,5.842,149.173
C09076=1171.955,-39.148,-43.970,179.551,5.841,149.174
C09077=1171.959,-39.398,-43.959,179.549,5.840,149.174
C09078=1171.965,-39.648,-43.947,179.546,5.840,149.175
C09079=1171.971,-39.897,-43.934,179.544,5.840,149.175
C09080=1171.976,-40.147,-43.923,179.542,5.839,149.176
C09081=1171.981,-40.396,-43.911,179.539,5.839,149.177
C09082=1171.986,-40.646,-43.899,179.537,5.838,149.177
C09083=1171.992,-40.896,-43.887,179.534,5.838,149.178
C09084=1171.996,-41.145,-43.875,179.532,5.837,149.179
C09085=1172.001,-41.395,-43.864,179.530,5.837,149.179
C09086=1172.007,-41.645,-43.852,179.527,5.837,149.180
C09087=1172.012,-41.895,-43.840,179.525,5.836,149.180
C09088=1172.017,-42.144,-43.829,179.523,5.836,149.181
C09089=1172.022,-42.394,-43.817,179.520,5.835,149.182
C09090=1172.028,-42.643,-43.806,179.518,5.835,149.182
C09091=1172.033,-42.893,-43.793,179.516,5.835,149.183
C09092=1172.038,-43.143,-43.781,179.513,5.834,149.183
C09093=1172.043,-43.392,-43.770,179.511,5.834,149.184
C09094=1172.048,-43.642,-43.758,179.508,5.833,149.185
C09095=1172.054,-43.892,-43.746,179.506,5.832,149.185
C09096=1172.059,-44.142,-43.735,179.504,5.833,149.186
C09097=1172.064,-44.392,-43.723,179.502,5.832,149.186
C09098=1172.069,-44.641,-43.712,179.499,5.831,149.187
C09099=1172.075,-44.890,-43.700,179.496,5.831,149.188
C09100=1172.080,-45.140,-43.688,179.494,5.830,149.188
C09101=1172.085,-45.390,-43.677,179.492,5.831,149.189
C09102=1172.090,-45.639,-43.664,179.489,5.830,149.190
C09103=1172.095,-45.889,-43.653,179.487,5.829,149.190
C09104=1172.100,-46.139,-43.641,179.485,5.829,149.191
C09105=1172.106,-46.388,-43.630,179.482,5.828,149.191
C09106=1172.111,-46.638,-43.618,179.480,5.829,149.192
C09107=1172.116,-46.888,-43.607,179.478,5.828,149.193
C09108=1172.121,-47.137,-43.595,179.475,5.827,149.193
C09109=1172.126,-47.387,-43.583,179.473,5.827,149.194
C09110=1172.131,-47.637,-43.572,179.471,5.826,149.194
C09111=1172.137,-47.886,-43.561,179.469,5.826,149.195
C09112=1172.142,-48.136,-43.549,179.466,5.826,149.196
C09113=1172.147,-48.386,-43.537,179.464,5.825,149.196
C09114=1172.153,-48.636,-43.526,179.461,5.825,149.197
C09115=1172.158,-48.886,-43.515,179.459,5.825,149.198
C09116=1172.164,-49.135,-43.503,179.457,5.824,149.198
C09117=1172.168,-49.385,-43.492,179.454,5.824,149.199
C09118=1172.174,-49.655,-43.479,179.452,5.823,149.199
C09119=1172.180,-49.925,-43.467,179.449,5.823,149.200
C09120=1172.185,-50.196,-43.454,179.447,5.822,149.201
C09121=1172.191,-50.467,-43.442,179.444,5.822,149.202
C09122=1172.196,-50.716,-43.431,179.442,5.821,149.202
C09123=1172.201,-50.966,-43.419,179.440,5.821,149.203
C09124=1172.206,-51.215,-43.408,179.437,5.821,149.203
C09125=1172.212,-51.465,-43.396,179.435,5.820,149.204
C09126=1172.216,-51.715,-43.385,179.432,5.820,149.205
C09127=1172.223,-51.965,-43.374,179.430,5.820,149.205
C09128=1172.227,-52.214,-43.363,179.428,5.819,149.206
C09129=1172.233,-52.464,-43.351,179.425,5.819,149.206
C09130=1172.237,-52.714,-43.340,179.423,5.818,149.207
C09131=1172.243,-52.963,-43.329,179.421,5.819,149.208
C09132=1172.248,-53.213,-43.317,179.419,5.818,149.208
C09133=1172.253,-53.463,-43.306,179.416,5.817,149.209
C09134=1172.259,-53.713,-43.294,179.413,5.817,149.210
C09135=1172.264,-53.962,-43.283,179.411,5.816,149.210
C09136=1172.269,-54.211,-43.272,179.409,5.816,149.211
C09137=1172.274,-54.461,-43.260,179.407,5.816,149.211
C09138=1172.280,-54.711,-43.250,179.404,5.815,149.212
C09139=1172.285,-54.961,-43.238,179.402,5.815,149.213
C09140=1172.290,-55.210,-43.227,179.400,5.815,149.213
C09141=1172.294,-55.460,-43.215,179.397,5.814,149.214
C09142=1172.301,-55.710,-43.205,179.395,5.814,149.214
C09143=1172.305,-55.960,-43.193,179.393,5.813,149.215
C09144=1172.310,-56.209,-43.182,179.390,5.814,149.216
C09145=1172.316,-56.458,-43.171,179.388,5.813,149.216
C09146=1172.321,-56.709,-43.160,179.386,5.812,149.217
C09147=1172.327,-56.959,-43.148,179.383,5.812,149.217
C09148=1172.331,-57.208,-43.137,179.381,5.812,149.218
C09149=1172.337,-57.458,-43.127,179.379,5.812,149.219
C09150=1172.342,-57.708,-43.115,179.376,5.811,149.219
C09151=1172.347,-57.957,-43.103,179.374,5.810,149.220
C09152=1172.352,-58.206,-43.093,179.372,5.810,149.220
C09153=1172.357,-58.456,-43.082,179.370,5.810,149.221
C09154=1172.363,-58.706,-43.070,179.367,5.809,149.222
C09155=1172.368,-58.955,-43.059,179.365,5.809,149.222
